// TIA Portal project "03_Montage_2018-09-26_KW" (V14)

(* hardware
DEVICE "S7300/ET200M-Station_4"  S7-300 station
   slot 0: "Profilschiene_0"  Rail  6ES7 390-1***0-0AA0
   slot 1: "PS 307 5A_1"  PS 307 5A  6ES7 307-1EA01-0AA0
   slot 2: "PLC_WBS_Bus"  CPU 314C-2 DP  6ES7 314-6CH04-0AB0  V3.3
      slot 0: "MPI-Schnittstelle_1"  MPI
      slot 1: "DP-Schnittstelle_1"  DP
      slot 2: "DI 24/DO 16_1"  DI24/DO16
      slot 3: "AI 5/AO 2_1"  AI5/AO2
      slot 4: "Zählen_1"  Counter
      slot 5: "Positionieren_1"  Positioning
   slot 4: "DI 64x24VDC sinking/souring_1"  DI64 x 24VDC  6ES7 321-1BP00-0AA0
   slot 5: "DI 64x24VDC sinking/souring_2"  DI64 x 24VDC  6ES7 321-1BP00-0AA0
   slot 6: "DI 64x24VDC sinking/souring_3"  DI64 x 24VDC  6ES7 321-1BP00-0AA0
   slot 7: "DI 64x24VDC sinking/souring_4"  DI64 x 24VDC  6ES7 321-1BP00-0AA0
   slot 8: "DO 64x24VDC/0.3A sourcing_1"  DO64 x 24VDC / 0.3A, P  6ES7 322-1BP00-0AA0
   slot 9: "DO 64x24VDC/0.3A sourcing_2"  DO64 x 24VDC / 0.3A, P  6ES7 322-1BP00-0AA0
   slot 10: "DO 64x24VDC/0.3A sourcing_3"  DO64 x 24VDC / 0.3A, P  6ES7 322-1BP00-0AA0
   slot 11: "DO 64x24VDC/0.3A sourcing_4"  DO64 x 24VDC / 0.3A, P  6ES7 322-1BP00-0AA0
*)

// ===== PLC "PLC_WBS_Bus"  CPU 314C-2 DP =====

VAR_GLOBAL   // PLC tag table "Standard-Variablentabelle"
   "Tag_1" AT %M20.0 : Bool;
   "Tag_2" AT %T0 : Timer;
END_VAR

VAR_GLOBAL   // PLC tag table "Betriebsart"
   "S0_HS" AT %E0.0 : Bool;   // Hauptschalter 0-Aus, 1-Ein
   "S1_Not_Halt" AT %E0.1 : Bool;   // Not-Halt NC
   "S2_START" AT %E0.2 : Bool;   // Taster START NO
   "S3_STOP" AT %E0.3 : Bool;   // Taster STOP NC
   "Res_E04" AT %E0.4 : Bool;
   "Res_E05" AT %E0.5 : Bool;
   "Res_E06" AT %E0.6 : Bool;
   "Res_E07" AT %E0.7 : Bool;
   "Res_E10" AT %E1.0 : Bool;
   "Res_E11" AT %E1.1 : Bool;
   "Res_E12" AT %E1.2 : Bool;
   "Res_E13" AT %E1.3 : Bool;
   "Res_E14" AT %E1.4 : Bool;
   "Res_E15" AT %E1.5 : Bool;
   "Res_E16" AT %E1.6 : Bool;
   "Factory_IO_RUN" AT %E1.7 : Bool;   // Rückmeldung Factory IO läuft
   "P1_MS_RT" AT %A0.0 : Bool;   // Meldesäule Rot
   "P2_MS_GE" AT %A0.1 : Bool;   // Meldesäule Gelb
   "P3_MS_GN" AT %A0.2 : Bool;   // Meldesäule Grün
   "P10_START" AT %A0.3 : Bool;   // Anzeige grün in START-Taster
   "P11_STOP" AT %A0.4 : Bool;   // Anzeige gelb in START-Taster
   "Res_A0.5" AT %A0.5 : Bool;
   "P12_Anfahrwarnung" AT %A0.6 : Bool;   // Rundumleuchte System
   "P13_Sirene" AT %A0.7 : Bool;   // Sirene System
   "Res_A10" AT %A1.0 : Bool;
   "Res_A11" AT %A1.1 : Bool;
   "Res_A12" AT %A1.2 : Bool;
   "Res_A13" AT %A1.3 : Bool;
   "Res_A14" AT %A1.4 : Bool;
   "Res_A15" AT %A1.5 : Bool;
   "Res_A16" AT %A1.6 : Bool;
   "Res_A17" AT %A1.7 : Bool;
   "Log_1" AT %M0.1 : Bool;   // statisch "1"
   "Log_0" AT %M0.0 : Bool;   // statisch "0"
   "Takt_1HZ" AT %M100.5 : Bool;   // Taktmerker 1 Hz
END_VAR

VAR_GLOBAL   // PLC tag table "Montage"
   "B3001_TB3001" AT %E2.0 : Bool;   // Transportband-Ende NC
   "B3002_TB3001" AT %E2.1 : Bool;   // Teil nachPositionierer NC
   "B3003_Teil_vor_POS" AT %E2.2 : Bool;   // Teil vor Positionierer NC
   "B3004_TB3001" AT %E2.3 : Bool;   // Transportband-Anfang NC
   "B3005_TB3002" AT %E2.4 : Bool;   // Transportband-Ende NC
   "B3006_TB3006" AT %E2.5 : Bool;   // Teil vor Schwenkarm NC
   "B3007_UT_BL" AT %E2.6 : Bool;   // Farbsensor Erkennung Farbteil Unterteil blau
   "B3008_OT_BL" AT %E2.7 : Bool;   // Farbsensor Erkennung Farbteil Oberteil blau
   "B3009_TB3006" AT %E3.0 : Bool;   // Transportband-Anfang NC
   "B3010_TB3007" AT %E3.1 : Bool;   // Transportband-Ende NC
   "B3011_TB3007" AT %E3.2 : Bool;   // Transportband-Anfang NC
   "B3012_TB3008" AT %E3.3 : Bool;   // Transportband-Ende NC
   "B3013_TB3008" AT %E3.4 : Bool;   // Transportband-Anfang NC
   "B3014_TB3005" AT %E3.5 : Bool;   // Transportband-Anfang NC
   "B3015_TB3005" AT %E3.6 : Bool;   // Transportband-Ende
   "B3016_TB3004" AT %E3.7 : Bool;   // Transportband-Anfang
   "B3017_Teil_vor_POS" AT %E4.0 : Bool;   // Teil vor Positionierer NC
   "B3018_TB3004" AT %E4.1 : Bool;   // Transportband-Ende NC
   "B3030_POS3001_geklemmt" AT %E4.2 : Bool;   // Positionierer RM geklemmt
   "B3031_POS3001_Heben_Senken" AT %E4.3 : Bool;   // Positionierer RM Bewegung
   "B3040_POS3002_geklemmt" AT %E4.4 : Bool;   // Positionierer RM geklemmt
   "B3041_POS3002_Heben_Senken" AT %E4.5 : Bool;   // Positionierer RM Bewegung
   "Res_E46" AT %E4.6 : Bool;
   "Res_E47" AT %E4.7 : Bool;
   "B3050_PAP3001_RM_X" AT %E5.0 : Bool;
   "B3051_PAP3001_RM_Z" AT %E5.1 : Bool;
   "B3052_PAP3001_Teil_erkannt" AT %E5.2 : Bool;
   "B3070_FZ_3001_Busy" AT %E5.3 : Bool;
   "B3071_FZ_3001_Error" AT %E5.4 : Bool;
   "B3072_FZ_Tür_offen" AT %E5.5 : Bool;
   "Res_E56" AT %E5.6 : Bool;
   "Res_E57" AT %E5.7 : Bool;
   "B4001_TB4001" AT %E6.0 : Bool;   // Transportband-Ende NC
   "B4002_TB4001" AT %E6.1 : Bool;   // Teil nachPositionierer NC
   "B4003_Teil_vor_POS" AT %E6.2 : Bool;   // Teil vor Positionierer NC
   "B4004_TB4001" AT %E6.3 : Bool;   // Transportband-Anfang NC
   "B4005_TB4002" AT %E6.4 : Bool;   // Transportband-Ende NC
   "B4006_TB4006" AT %E6.5 : Bool;   // Teil vor Schwenkarm NC
   "B4007_UT_GN" AT %E6.6 : Bool;   // Farbsensor Erkennung Farbteil Unterteil grün
   "B4008_OT_GN" AT %E6.7 : Bool;   // Farbsensor Erkennung Farbteil Oberteil grün
   "B4009_TB4006" AT %E7.0 : Bool;   // Transportband-Anfang NC
   "B4010_TB4007" AT %E7.1 : Bool;   // Transportband-Ende NC
   "B4011_TB4007" AT %E7.2 : Bool;   // Transportband-Anfang NC
   "B4012_TB4008" AT %E7.3 : Bool;   // Transportband-Ende NC
   "B4013_TB4008" AT %E7.4 : Bool;   // Transportband-Anfang NC
   "B4014_TB4005" AT %E7.5 : Bool;   // Transportband-Anfang NC
   "B4015_TB4005" AT %E7.6 : Bool;   // Transportband-Ende
   "B4016_TB4004" AT %E7.7 : Bool;   // Transportband-Anfang
   "B4017_Teil_vor_POS" AT %E8.0 : Bool;   // Teil vor Positionierer NC
   "B4018_TB4004" AT %E8.1 : Bool;   // Transportband-Ende NC
   "B4030_POS4001_geklemmt" AT %E8.2 : Bool;   // Positionierer RM geklemmt
   "B4031_POS4001_Heben_Senken" AT %E8.3 : Bool;   // Positionierer RM Bewegung
   "B4040_POS4002_geklemmt" AT %E8.4 : Bool;   // Positionierer RM geklemmt
   "B4041_POS4002_Heben_Senken" AT %E8.5 : Bool;   // Positionierer RM Bewegung
   "Res_E86" AT %E8.6 : Bool;
   "Res_E87" AT %E8.7 : Bool;
   "B4050_PAP4001_RM_X" AT %E9.0 : Bool;   // Pick-and-Place X-aktiv
   "B4051_PAP4001_RM_Z" AT %E9.1 : Bool;   // Pick-and-Place Z-aktiv
   "B4052_PAP4001_Teil_erkannt" AT %E9.2 : Bool;   // Teil am Greifer erkannt
   "B4070_FZ_4001_Busy" AT %E9.3 : Bool;   // Fertigungszentrum
   "B4071_FZ_4001_Error" AT %E9.4 : Bool;   // Fertigungszentrum
   "B4072_FZ_4001_Tür_offen" AT %E9.5 : Bool;   // Fertigungszentrum
   "Res_E96" AT %E9.6 : Bool;
   "Res_E97" AT %E9.7 : Bool;
   "TB3001" AT %A2.0 : Bool;
   "TB3002" AT %A2.1 : Bool;
   "TB3003" AT %A2.2 : Bool;
   "TB3004" AT %A2.3 : Bool;
   "TB3005" AT %A2.4 : Bool;
   "TB3006" AT %A2.5 : Bool;
   "TB3007" AT %A2.6 : Bool;
   "TB3008" AT %A2.7 : Bool;
   "FZ_3001_Start" AT %A3.0 : Bool;   // Fertigungszentrum Start
   "FZ_3001_Stop" AT %A3.1 : Bool;   // Fertigungszentrum Stop
   "FZ_3001_OT_UT" AT %A3.2 : Bool;   // Fertigungszentrum UT =0 / OT=1
   "Sorter_Arm_3001_schwenken" AT %A3.3 : Bool;
   "Sorter_Arm_3001_Band_V" AT %A3.4 : Bool;
   "Sorter_Arm_3001_Band_R" AT %A3.5 : Bool;
   "POS3001_Klemmen" AT %A3.6 : Bool;
   "POS3001_Heben" AT %A3.7 : Bool;
   "POS3002_Klemmen" AT %A4.0 : Bool;
   "POS3002_Heben" AT %A4.1 : Bool;
   "PAP3001_X" AT %A4.2 : Bool;
   "PAP3001_Z" AT %A4.3 : Bool;
   "PAP3001_Greifer" AT %A4.4 : Bool;
   "STOP_3001" AT %A4.5 : Bool;
   "Res_A46" AT %A4.6 : Bool;
   "Emitter_1" AT %A4.7 : Bool;
   "TB4001" AT %A5.0 : Bool;
   "TB4002" AT %A5.1 : Bool;
   "TB4003" AT %A5.2 : Bool;
   "TB4004" AT %A5.3 : Bool;
   "TB4005" AT %A5.4 : Bool;
   "TB4006" AT %A5.5 : Bool;
   "TB4007" AT %A5.6 : Bool;
   "TB4008" AT %A5.7 : Bool;
   "FZ_4001_Start" AT %A6.0 : Bool;   // Fertigungszentrum Start
   "FZ_4001_Stop" AT %A6.1 : Bool;   // Fertigungszentrum Stop
   "FZ_4001_OT_UT" AT %A6.2 : Bool;   // Fertigungszentrum UT =0 / OT=1
   "Sorter_Arm_4001_schwenken" AT %A6.3 : Bool;
   "Sorter_Arm_4001_Band_V" AT %A6.4 : Bool;
   "Sorter_Arm_4001_Band_R" AT %A6.5 : Bool;
   "POS4001_Klemmen" AT %A6.6 : Bool;
   "POS4001_Heben" AT %A6.7 : Bool;
   "POS4002_Klemmen" AT %A7.0 : Bool;
   "POS4002_Heben" AT %A7.1 : Bool;
   "PAP4001_X" AT %A7.2 : Bool;
   "PAP4001_Z" AT %A7.3 : Bool;
   "PAP4001_Greifer" AT %A7.4 : Bool;
   "STOP4001" AT %A7.5 : Bool;
   "Res_A76" AT %A7.6 : Bool;
   "Emitter_2" AT %A7.7 : Bool;
   "FZ_3001_Bearbeitungszeit" AT %EW20 : Int;
   "FZ_4001_Bearbeitungszeit" AT %EW22 : Int;
END_VAR

VAR_GLOBAL   // PLC tag table "KW"
   "Anlage_Start" AT %M22.0 : Bool;
   "Freigabe_Start" AT %M22.1 : Bool;
   "M_HOT_HALT" AT %M22.2 : Bool;
   "FLK_S2_Start" AT %M22.3 : Bool;
   "B1_Freigabe" AT %M22.4 : Bool;
   "Teile_Typ" AT %M22.5 : Bool;
   "FLK_B4010_TB4007" AT %M22.6 : Bool;
   "FreiFürTB4006" AT %M22.7 : Bool;
   "UT_an_Weiche" AT %M23.0 : Bool;
   "OT_an_Weiche" AT %M23.1 : Bool;
   "FreiFürTB4005" AT %M23.2 : Bool;
   "Glob_Sperre" AT %M23.3 : Bool;
   "FreiFürTB4002" AT %M23.4 : Bool;
   "M_Entklemmen" AT %M23.5 : Bool;
   "03_M_OT_Abfuehren" AT %M23.6 : Bool;
   "03_M_UT_Abfuehren" AT %M23.7 : Bool;
   "MT_OT_Bereit" AT %M24.0 : Bool;
   "MT_UT_Bereit" AT %M24.1 : Bool;
   "03_GRN_OT_det" AT %M24.2 : Bool;
   "03_GRN_UT_det" AT %M24.3 : Bool;
   "03_BLAU_OT_det" AT %M24.4 : Bool;
   "03_BLAU_UT_det" AT %M24.5 : Bool;
   "03_GRN_FRGB_CNC" AT %M24.6 : Bool;
   "03_BLAU_FRGB_CNC" AT %M24.7 : Bool;
   "03_GRN_CNC_MTR_AN" AT %M25.0 : Bool;
   "03_BLAU_CNC_MTR_AN" AT %M25.1 : Bool;
   "delete_1" AT %M25.2 : Bool;
   "delete_2" AT %M25.3 : Bool;
   "03_GRN_OT_FRG" AT %M25.4 : Bool;
   "03_GRN_UT_FRG" AT %M25.5 : Bool;
   "03_BLAU_OT_FRG" AT %M25.6 : Bool;
   "03_BLAU_UT_FRG" AT %M25.7 : Bool;
END_VAR

DATA_BLOCK "03_04-OT_Grueneteile"   // DB2
{ S7_Optimized_Access := 'FALSE' }
VERSION : 0.1
// stored: InstanceOfName Foerderband_m_Klemme
"Foerderband_m_Klemme"
BEGIN
END_DATA_BLOCK

DATA_BLOCK "03_04_UT_Grueneteile"   // DB3
{ S7_Optimized_Access := 'FALSE' }
VERSION : 0.1
// stored: InstanceOfName Foerderband_m_Klemme
"Foerderband_m_Klemme"
BEGIN
END_DATA_BLOCK

DATA_BLOCK "03_04_PnP_Grueneteile"   // DB4
{ S7_Optimized_Access := 'FALSE' }
VERSION : 0.1
// stored: InstanceOfName Pick_n_Place
"Pick_n_Place"
BEGIN
END_DATA_BLOCK

DATA_BLOCK "03_04_MNTG_Grueneteile"   // DB5
{ S7_Optimized_Access := 'FALSE' }
VERSION : 0.1
// stored: InstanceOfName 03_04_MNTG_BL
"03_04_MNTG_BL"
BEGIN
END_DATA_BLOCK

DATA_BLOCK "03_04_MNTG_Blaueteile"   // DB6
{ S7_Optimized_Access := 'FALSE' }
VERSION : 0.1
// stored: InstanceOfName 03_04_MNTG_BL
"03_04_MNTG_BL"
BEGIN
END_DATA_BLOCK

DATA_BLOCK "03_04-OT_Blaueteile"   // DB7
{ S7_Optimized_Access := 'FALSE' }
VERSION : 0.1
// stored: InstanceOfName Foerderband_m_Klemme
"Foerderband_m_Klemme"
BEGIN
END_DATA_BLOCK

DATA_BLOCK "03_04_UT_Blaueteile"   // DB8
{ S7_Optimized_Access := 'FALSE' }
VERSION : 0.1
// stored: InstanceOfName Foerderband_m_Klemme
"Foerderband_m_Klemme"
BEGIN
END_DATA_BLOCK

DATA_BLOCK "03_04_PnP_Blaueteile"   // DB9
{ S7_Optimized_Access := 'FALSE' }
VERSION : 0.1
// stored: InstanceOfName Pick_n_Place
"Pick_n_Place"
BEGIN
END_DATA_BLOCK

DATA_BLOCK "FB_OT_Gruen"   // DB10
{ S7_Optimized_Access := 'FALSE' }
VERSION : 0.1
// stored: InstanceOfName Foerderband_m_Klemme
"Foerderband_m_Klemme"
BEGIN
END_DATA_BLOCK

DATA_BLOCK "FB_UT_Gruen"   // DB11
{ S7_Optimized_Access := 'FALSE' }
VERSION : 0.1
// stored: InstanceOfName Foerderband_m_Klemme
"Foerderband_m_Klemme"
BEGIN
END_DATA_BLOCK

DATA_BLOCK "03_01_Grueneteile"   // DB12
{ S7_Optimized_Access := 'FALSE' }
VERSION : 0.1
// stored: InstanceOfName 03_01_Anlaufbaender
"03_01_Anlaufbaender"
BEGIN
END_DATA_BLOCK

DATA_BLOCK "03_01_Blaueteile"   // DB13
{ S7_Optimized_Access := 'FALSE' }
VERSION : 0.1
// stored: InstanceOfName 03_01_Anlaufbaender
"03_01_Anlaufbaender"
BEGIN
END_DATA_BLOCK

DATA_BLOCK "03_02_Grueneteile"   // DB14
{ S7_Optimized_Access := 'FALSE' }
VERSION : 0.1
// stored: InstanceOfName 03_02_Bearbeitungszelle
"03_02_Bearbeitungszelle"
BEGIN
END_DATA_BLOCK

DATA_BLOCK "03_02_Blaueteile"   // DB15
{ S7_Optimized_Access := 'FALSE' }
VERSION : 0.1
// stored: InstanceOfName 03_02_Bearbeitungszelle
"03_02_Bearbeitungszelle"
BEGIN
END_DATA_BLOCK

DATA_BLOCK "03_03_Grueneteile"   // DB16
{ S7_Optimized_Access := 'FALSE' }
VERSION : 0.1
// stored: InstanceOfName 03_03_Weiche
"03_03_Weiche"
BEGIN
END_DATA_BLOCK

DATA_BLOCK "03_03_Blaueteile"   // DB17
{ S7_Optimized_Access := 'FALSE' }
VERSION : 0.1
// stored: InstanceOfName 03_03_Weiche
"03_03_Weiche"
BEGIN
END_DATA_BLOCK

DATA_BLOCK "PnP_Gruen"   // DB18
{ S7_Optimized_Access := 'FALSE' }
VERSION : 0.1
// stored: InstanceOfName Pick_n_Place
"Pick_n_Place"
BEGIN
END_DATA_BLOCK

DATA_BLOCK "03_04_MNTG_GR_DB"   // DB19
{ S7_Optimized_Access := 'FALSE' }
VERSION : 0.1
// stored: InstanceOfName 03_04_MNTG_GR
"03_04_MNTG_GR"
BEGIN
END_DATA_BLOCK

FUNCTION_BLOCK "03_04_MNTG_BL"   // FB1, FBD
{ S7_Optimized_Access := 'FALSE' }
VERSION : 0.1
   VAR_OUTPUT
      OT_Freigabe : Bool;
      UT_Freigabe : Bool;
   END_VAR
   VAR
      OT_angesaugt : Bool;
      OT_losgelassen : Bool;
      OT_Band : "Foerderband_m_Klemme";
      UT_Band : "Foerderband_m_Klemme";
      PicknPlace : "Pick_n_Place";
   END_VAR
BEGIN

REGION Network 1: BLAU OT Klemm-Foerderband
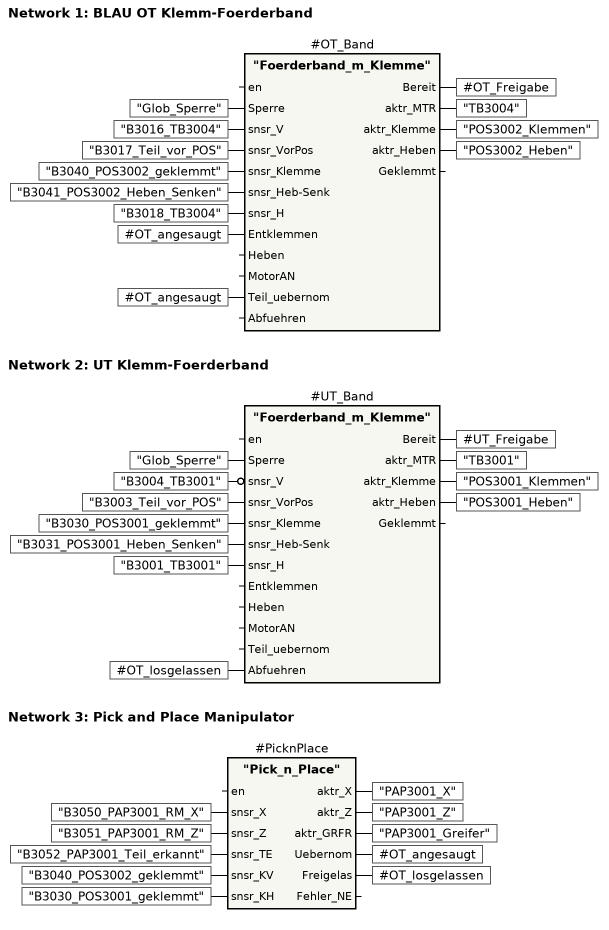
   #OT_Band(Sperre := "Glob_Sperre",   // "Foerderband_m_Klemme"
            snsr_V := "B3016_TB3004",
            snsr_VorPos := "B3017_Teil_vor_POS",
            snsr_Klemme := "B3040_POS3002_geklemmt",
            "snsr_Heb-Senk" := "B3041_POS3002_Heben_Senken",
            snsr_H := "B3018_TB3004",
            Entklemmen := #OT_angesaugt,
            Teil_uebernom := #OT_angesaugt,
            Bereit => #OT_Freigabe,
            aktr_MTR => "TB3004",
            aktr_Klemme => "POS3002_Klemmen",
            aktr_Heben => "POS3002_Heben");
END_REGION

REGION Network 2: UT Klemm-Foerderband
   #UT_Band(Sperre := "Glob_Sperre",   // "Foerderband_m_Klemme"
            snsr_V := NOT "B3004_TB3001",
            snsr_VorPos := "B3003_Teil_vor_POS",
            snsr_Klemme := "B3030_POS3001_geklemmt",
            "snsr_Heb-Senk" := "B3031_POS3001_Heben_Senken",
            snsr_H := "B3001_TB3001",
            Abfuehren := #OT_losgelassen,
            Bereit => #UT_Freigabe,
            aktr_MTR => "TB3001",
            aktr_Klemme => "POS3001_Klemmen",
            aktr_Heben => "POS3001_Heben");
END_REGION

REGION Network 3: Pick and Place Manipulator
   #PicknPlace(snsr_X := "B3050_PAP3001_RM_X",   // "Pick_n_Place"
               snsr_Z := "B3051_PAP3001_RM_Z",
               snsr_TE := "B3052_PAP3001_Teil_erkannt",
               snsr_KV := "B3040_POS3002_geklemmt",
               snsr_KH := "B3030_POS3001_geklemmt",
               aktr_X => "PAP3001_X",
               aktr_Z => "PAP3001_Z",
               aktr_GRFR => "PAP3001_Greifer",
               Uebernom => #OT_angesaugt,
               Freigelas => #OT_losgelassen);
END_REGION
END_FUNCTION_BLOCK

FUNCTION_BLOCK "03_04_MNTG_GR"   // FB2, FBD
{ S7_Optimized_Access := 'FALSE' }
VERSION : 0.1
   VAR_OUTPUT
      OT_Freigabe : Bool;
      UT_Freigabe : Bool;
   END_VAR
   VAR
      OT_Band_DB : "Foerderband_m_Klemme";
      UT_Band_DB : "Foerderband_m_Klemme";
      PnP_DB : "Pick_n_Place";
      OT_angesaugt : Bool;
      OT_losgelassen : Bool;
   END_VAR
BEGIN

REGION Network 1: GRUEN OT Klemm-Foerderband
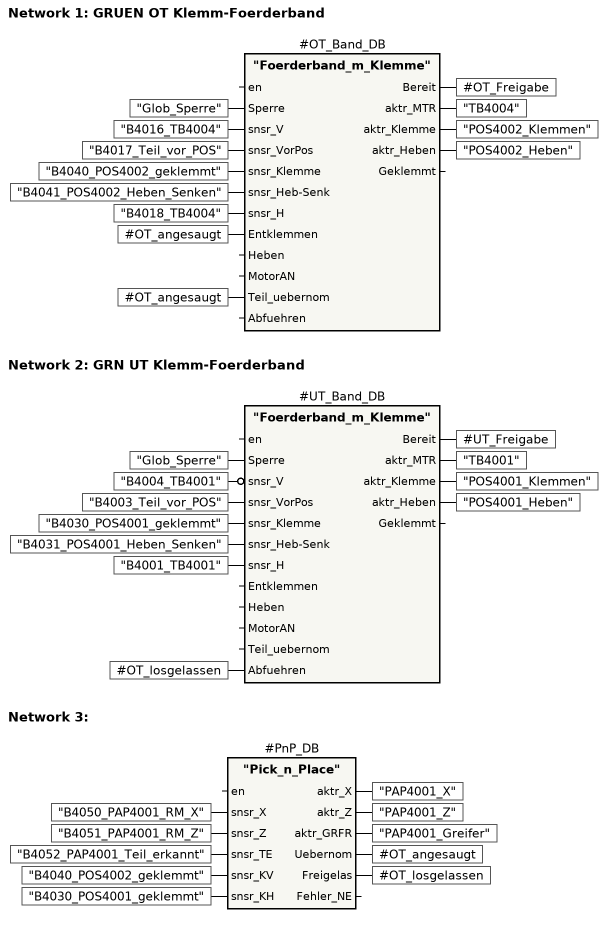
   #OT_Band_DB(Sperre := "Glob_Sperre",   // "Foerderband_m_Klemme"
               snsr_V := "B4016_TB4004",
               snsr_VorPos := "B4017_Teil_vor_POS",
               snsr_Klemme := "B4040_POS4002_geklemmt",
               "snsr_Heb-Senk" := "B4041_POS4002_Heben_Senken",
               snsr_H := "B4018_TB4004",
               Entklemmen := #OT_angesaugt,
               Teil_uebernom := #OT_angesaugt,
               Bereit => #OT_Freigabe,
               aktr_MTR => "TB4004",
               aktr_Klemme => "POS4002_Klemmen",
               aktr_Heben => "POS4002_Heben");
END_REGION

REGION Network 2: GRN UT Klemm-Foerderband
   #UT_Band_DB(Sperre := "Glob_Sperre",   // "Foerderband_m_Klemme"
               snsr_V := NOT "B4004_TB4001",
               snsr_VorPos := "B4003_Teil_vor_POS",
               snsr_Klemme := "B4030_POS4001_geklemmt",
               "snsr_Heb-Senk" := "B4031_POS4001_Heben_Senken",
               snsr_H := "B4001_TB4001",
               Abfuehren := #OT_losgelassen,
               Bereit => #UT_Freigabe,
               aktr_MTR => "TB4001",
               aktr_Klemme => "POS4001_Klemmen",
               aktr_Heben => "POS4001_Heben");
END_REGION

REGION Network 3
   #PnP_DB(snsr_X := "B4050_PAP4001_RM_X",   // "Pick_n_Place"
           snsr_Z := "B4051_PAP4001_RM_Z",
           snsr_TE := "B4052_PAP4001_Teil_erkannt",
           snsr_KV := "B4040_POS4002_geklemmt",
           snsr_KH := "B4030_POS4001_geklemmt",
           aktr_X => "PAP4001_X",
           aktr_Z => "PAP4001_Z",
           aktr_GRFR => "PAP4001_Greifer",
           Uebernom => #OT_angesaugt,
           Freigelas => #OT_losgelassen);
END_REGION
END_FUNCTION_BLOCK

FUNCTION_BLOCK "Foerderband_m_Klemme"   // FB3, LAD
{ S7_Optimized_Access := 'FALSE' }
VERSION : 0.1
   VAR_INPUT
      Sperre : Bool;
      snsr_V : Bool;   // (NC) =1 wenn betätigt
      snsr_VorPos : Bool;   // (NO) =0 wenn betätigt
      snsr_Klemme : Bool;   // (NC) =1 wenn betätigt
      "snsr_Heb-Senk" : Bool;   // (NO) =0 wenn betätigt
      snsr_H : Bool;   // (NO) =0 wenn betätigt
      Entklemmen : Bool;   // =1 entklemmen
      Heben : Bool;   // =0 unten, =1 oben
      MotorAN : Bool;   // =1 Motor AN, =0 Motor AUS
      Teil_uebernom : Bool;   // =0 passiv, =1 aktiv
   END_VAR
   VAR_OUTPUT
      Bereit : Bool;
      aktr_MTR : Bool;
      aktr_Klemme : Bool;
      aktr_Heben : Bool;
      Geklemmt : Bool;
   END_VAR
   VAR_IN_OUT
      Abfuehren : Bool;
   END_VAR
   VAR
      Beladen : Bool;
      FLK_Letzter_Sensor : Bool;
      "FLK_Vor-Pos" : Bool;
      LetSens_P_Flanke : Bool;
      Abfuhr_Modus : Bool;
   END_VAR
   VAR_TEMP   // added for the SCL form of the ladder/FBD networks
      _w1 : Bool;
   END_VAR
BEGIN

REGION Network 1: Letzter Sensor positive Flankenerkennung
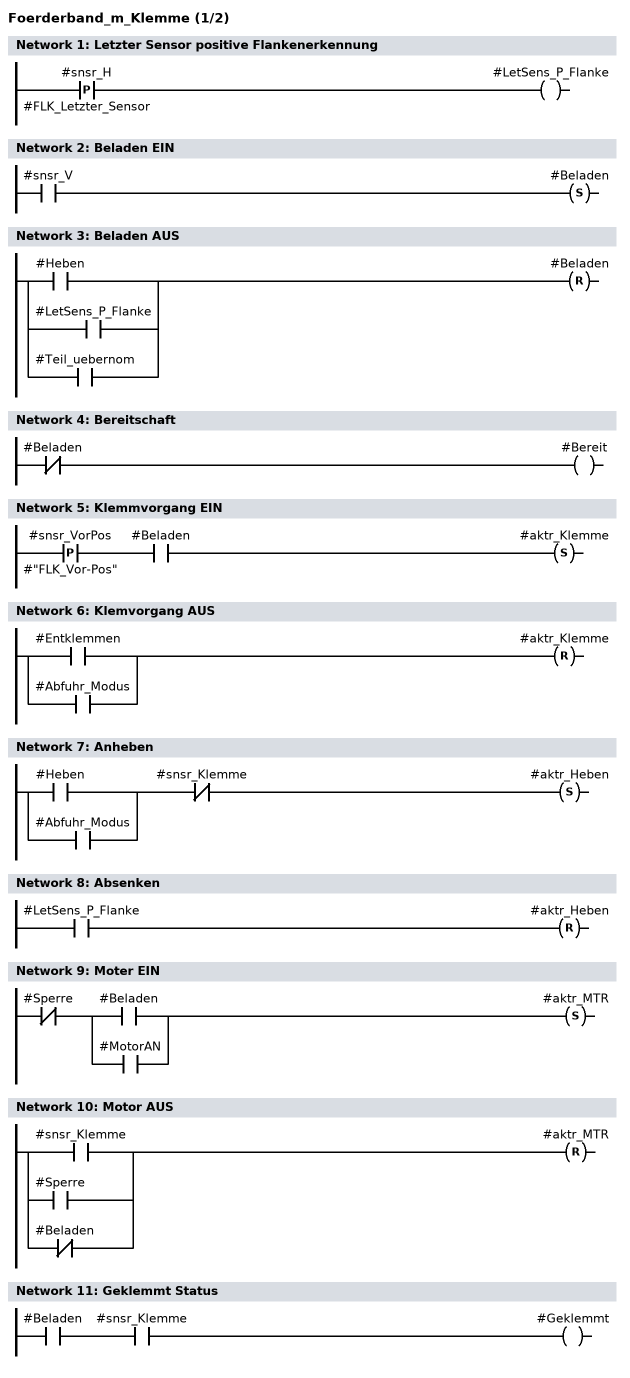
   RUNG wire#powerrail
      P_Contact(operand := #snsr_H, bit := #FLK_Letzter_Sensor)
      Coil( #LetSens_P_Flanke )
   END_RUNG
   // the same network as SCL:
   #_w1 := #snsr_H AND NOT #FLK_Letzter_Sensor;   // rising edge of #snsr_H
   #FLK_Letzter_Sensor := #snsr_H;
   #LetSens_P_Flanke := #_w1;
END_REGION

REGION Network 2: Beladen EIN
   RUNG wire#powerrail
      Contact( #snsr_V )
      S_Coil( #Beladen )
   END_RUNG
   // the same network as SCL:
   IF #snsr_V THEN #Beladen := TRUE; END_IF;
END_REGION

REGION Network 3: Beladen AUS
   RUNG wire#powerrail
      Contact( #Heben )
      wire#w1
      R_Coil( #Beladen )
   END_RUNG
   RUNG wire#powerrail
      Contact( #LetSens_P_Flanke )
   END_RUNG wire#w1
   RUNG wire#powerrail
      Contact( #Teil_uebernom )
   END_RUNG wire#w1
   // the same network as SCL:
   IF #Heben OR #LetSens_P_Flanke OR #Teil_uebernom THEN #Beladen := FALSE; END_IF;
END_REGION

REGION Network 4: Bereitschaft
   RUNG wire#powerrail
      I_Contact( #Beladen )
      Coil( #Bereit )
   END_RUNG
   // the same network as SCL:
   #Bereit := NOT #Beladen;
END_REGION

REGION Network 5: Klemmvorgang EIN
   RUNG wire#powerrail
      P_Contact(operand := #snsr_VorPos, bit := #"FLK_Vor-Pos")
      Contact( #Beladen )
      S_Coil( #aktr_Klemme )
   END_RUNG
   // the same network as SCL:
   #_w1 := #snsr_VorPos AND NOT #"FLK_Vor-Pos";   // rising edge of #snsr_VorPos
   #"FLK_Vor-Pos" := #snsr_VorPos;
   IF #_w1 AND #Beladen THEN #aktr_Klemme := TRUE; END_IF;
END_REGION

REGION Network 6: Klemvorgang AUS
   RUNG wire#powerrail
      Contact( #Entklemmen )
      wire#w1
      R_Coil( #aktr_Klemme )
   END_RUNG
   RUNG wire#powerrail
      Contact( #Abfuhr_Modus )
   END_RUNG wire#w1
   // the same network as SCL:
   IF #Entklemmen OR #Abfuhr_Modus THEN #aktr_Klemme := FALSE; END_IF;
END_REGION

REGION Network 7: Anheben
   RUNG wire#powerrail
      Contact( #Heben )
      wire#w1
      I_Contact( #snsr_Klemme )
      S_Coil( #aktr_Heben )
   END_RUNG
   RUNG wire#powerrail
      Contact( #Abfuhr_Modus )
   END_RUNG wire#w1
   // the same network as SCL:
   IF (#Heben OR #Abfuhr_Modus) AND NOT #snsr_Klemme THEN #aktr_Heben := TRUE; END_IF;
END_REGION

REGION Network 8: Absenken
   RUNG wire#powerrail
      Contact( #LetSens_P_Flanke )
      R_Coil( #aktr_Heben )
   END_RUNG
   // the same network as SCL:
   IF #LetSens_P_Flanke THEN #aktr_Heben := FALSE; END_IF;
END_REGION

REGION Network 9: Moter EIN
   RUNG wire#powerrail
      I_Contact( #Sperre )
      wire#w1
      Contact( #Beladen )
      wire#w2
      S_Coil( #aktr_MTR )
   END_RUNG
   RUNG wire#w1
      Contact( #MotorAN )
   END_RUNG wire#w2
   // the same network as SCL:
   IF NOT #Sperre AND (#Beladen OR #MotorAN) THEN #aktr_MTR := TRUE; END_IF;
END_REGION

REGION Network 10: Motor AUS
   RUNG wire#powerrail
      Contact( #snsr_Klemme )
      wire#w1
      R_Coil( #aktr_MTR )
   END_RUNG
   RUNG wire#powerrail
      Contact( #Sperre )
   END_RUNG wire#w1
   RUNG wire#powerrail
      I_Contact( #Beladen )
   END_RUNG wire#w1
   // the same network as SCL:
   IF #snsr_Klemme OR #Sperre OR NOT #Beladen THEN #aktr_MTR := FALSE; END_IF;
END_REGION

REGION Network 11: Geklemmt Status
   RUNG wire#powerrail
      Contact( #Beladen )
      Contact( #snsr_Klemme )
      Coil( #Geklemmt )
   END_RUNG
   // the same network as SCL:
   #Geklemmt := #Beladen AND #snsr_Klemme;
END_REGION

REGION Network 12: SR Abfuhr_Modus
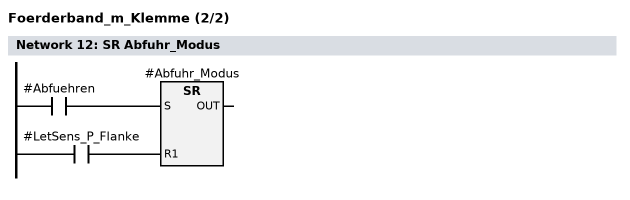
   RUNG wire#powerrail
      Contact( #Abfuehren )
      S_SR(operand := #Abfuhr_Modus, r1 := wire#w1)
   END_RUNG
   RUNG wire#powerrail
      Contact( #LetSens_P_Flanke )
   END_RUNG wire#w1
   // the same network as SCL:
   IF #Abfuehren THEN
       #Abfuhr_Modus := TRUE;   // SR flip-flop
   END_IF;
   IF #LetSens_P_Flanke THEN #Abfuhr_Modus := FALSE; END_IF;
END_REGION
END_FUNCTION_BLOCK

FUNCTION_BLOCK "03_01_Anlaufbaender"   // FB4, LAD
{ S7_Optimized_Access := 'FALSE' }
VERSION : 0.1
   VAR_INPUT
      snsr_V1 : Bool;
      snsr_V2 : Bool;
      snsr_H1 : Bool;
      snsr_H2 : Bool;
      Freigabe_IN : Bool;
      Sperre : Bool;
   END_VAR
   VAR_OUTPUT
      aktr_MTR_1 : Bool;
      aktr_MTR_2 : Bool;
      Freigabe_OUT : Bool;
   END_VAR
   VAR
      Beladen_1 : Bool;
      Beladen_2 : Bool;
      FLK_H1 : Bool;
      FLK_H2 : Bool;
   END_VAR
   VAR_TEMP   // added for the SCL form of the ladder/FBD networks
      _w1 : Bool;
   END_VAR
BEGIN

REGION Network 1: Reset Beladen_1
   // Reset des Statuses BELADEN der ersten Förderband
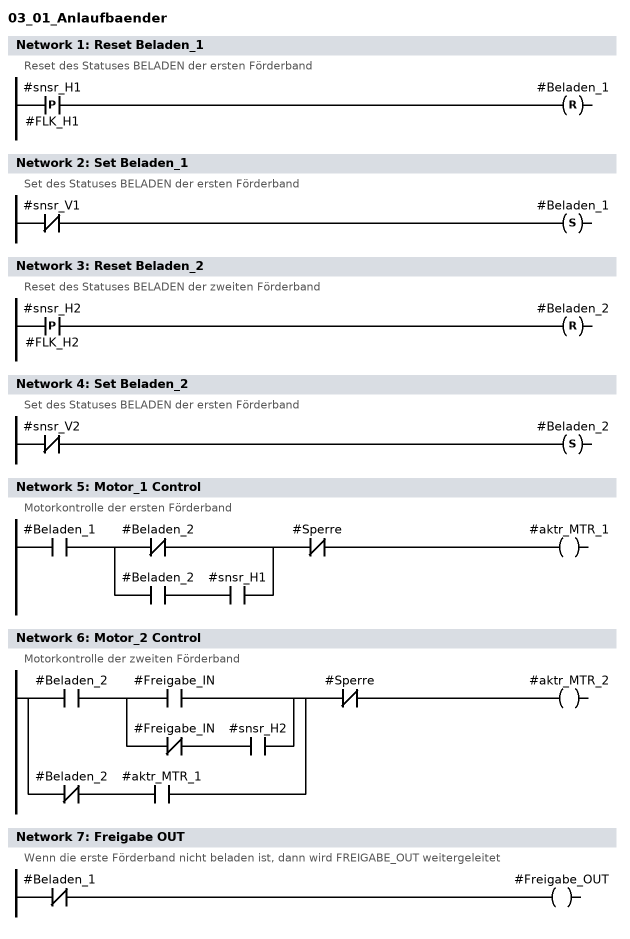
   RUNG wire#powerrail
      P_Contact(operand := #snsr_H1, bit := #FLK_H1)
      R_Coil( #Beladen_1 )
   END_RUNG
   // the same network as SCL:
   #_w1 := #snsr_H1 AND NOT #FLK_H1;   // rising edge of #snsr_H1
   #FLK_H1 := #snsr_H1;
   IF #_w1 THEN #Beladen_1 := FALSE; END_IF;
END_REGION

REGION Network 2: Set Beladen_1
   // Set des Statuses BELADEN der ersten Förderband
   RUNG wire#powerrail
      I_Contact( #snsr_V1 )
      S_Coil( #Beladen_1 )
   END_RUNG
   // the same network as SCL:
   IF NOT #snsr_V1 THEN #Beladen_1 := TRUE; END_IF;
END_REGION

REGION Network 3: Reset Beladen_2
   // Reset des Statuses BELADEN der zweiten Förderband
   RUNG wire#powerrail
      P_Contact(operand := #snsr_H2, bit := #FLK_H2)
      R_Coil( #Beladen_2 )
   END_RUNG
   // the same network as SCL:
   #_w1 := #snsr_H2 AND NOT #FLK_H2;   // rising edge of #snsr_H2
   #FLK_H2 := #snsr_H2;
   IF #_w1 THEN #Beladen_2 := FALSE; END_IF;
END_REGION

REGION Network 4: Set Beladen_2
   // Set des Statuses BELADEN der ersten Förderband
   RUNG wire#powerrail
      I_Contact( #snsr_V2 )
      S_Coil( #Beladen_2 )
   END_RUNG
   // the same network as SCL:
   IF NOT #snsr_V2 THEN #Beladen_2 := TRUE; END_IF;
END_REGION

REGION Network 5: Motor_1 Control
   // Motorkontrolle der ersten Förderband
   RUNG wire#powerrail
      Contact( #Beladen_1 )
      wire#w1
      I_Contact( #Beladen_2 )
      wire#w2
      I_Contact( #Sperre )
      Coil( #aktr_MTR_1 )
   END_RUNG
   RUNG wire#w1
      Contact( #Beladen_2 )
      Contact( #snsr_H1 )
   END_RUNG wire#w2
   // the same network as SCL:
   #aktr_MTR_1 := #Beladen_1 AND (NOT #Beladen_2 OR (#Beladen_2 AND #snsr_H1)) AND NOT #Sperre;
END_REGION

REGION Network 6: Motor_2 Control
   // Motorkontrolle der zweiten Förderband
   RUNG wire#powerrail
      Contact( #Beladen_2 )
      wire#w1
      Contact( #Freigabe_IN )
      wire#w2
      I_Contact( #Sperre )
      Coil( #aktr_MTR_2 )
   END_RUNG
   RUNG wire#w1
      I_Contact( #Freigabe_IN )
      Contact( #snsr_H2 )
   END_RUNG wire#w2
   RUNG wire#powerrail
      I_Contact( #Beladen_2 )
      Contact( #aktr_MTR_1 )
   END_RUNG wire#w2
   // the same network as SCL:
   #aktr_MTR_2 := ((#Beladen_2 AND (#Freigabe_IN OR (NOT #Freigabe_IN AND #snsr_H2))) OR (NOT #Beladen_2 AND #aktr_MTR_1)) AND NOT #Sperre;
END_REGION

REGION Network 7: Freigabe OUT
   // Wenn die erste Förderband nicht beladen ist, dann wird FREIGABE_OUT weitergeleitet
   RUNG wire#powerrail
      I_Contact( #Beladen_1 )
      Coil( #Freigabe_OUT )
   END_RUNG
   // the same network as SCL:
   #Freigabe_OUT := NOT #Beladen_1;
END_REGION
END_FUNCTION_BLOCK

FUNCTION_BLOCK "Pick_n_Place"   // FB5, LAD
TITLE = Montage Pick_n_Place
{ S7_Optimized_Access := 'FALSE' }
VERSION : 0.1
   VAR_INPUT
      snsr_X : Bool;
      snsr_Z : Bool;
      snsr_TE : Bool;
      snsr_KV : Bool;
      snsr_KH : Bool;
   END_VAR
   VAR_OUTPUT
      aktr_X : Bool;
      aktr_Z : Bool;
      aktr_GRFR : Bool;
      Uebernom : Bool;
      Freigelas : Bool;
      Fehler_NE : Bool;
   END_VAR
   VAR
      X0 : Bool;
      X1 : Bool;
      X2 : Bool;
      X3 : Bool;
      X4 : Bool;
      X5 : Bool;
      X6 : Bool;
      X7 : Bool;
      X8 : Bool;
      X9 : Bool;
      IF_X1 : Bool;
      IF_X2 : Bool;
      IF_X3 : Bool;
      IF_X4 : Bool;
      IF_X5 : Bool;
      IF_X6 : Bool;
      IF_X7 : Bool;
      IF_X8 : Bool;
      IF_X9 : Bool;
      flk_X1 : Bool;
      flk_X2 : Bool;
      flk_X3 : Bool;
      flk_X4 : Bool;
      flk_X5 : Bool;
      flk_X6 : Bool;
      flk_X7 : Bool;
      flk_X8 : Bool;
      flk_X9 : Bool;
      Zmove_ended : Bool;
      Xmove_ended : Bool;
      flk_Xmove : Bool;
      flk_Zmove : Bool;
   END_VAR
   VAR_TEMP   // added for the SCL form of the ladder/FBD networks
      _w1 : Bool;
   END_VAR
BEGIN

REGION Network 1: Grundstellung
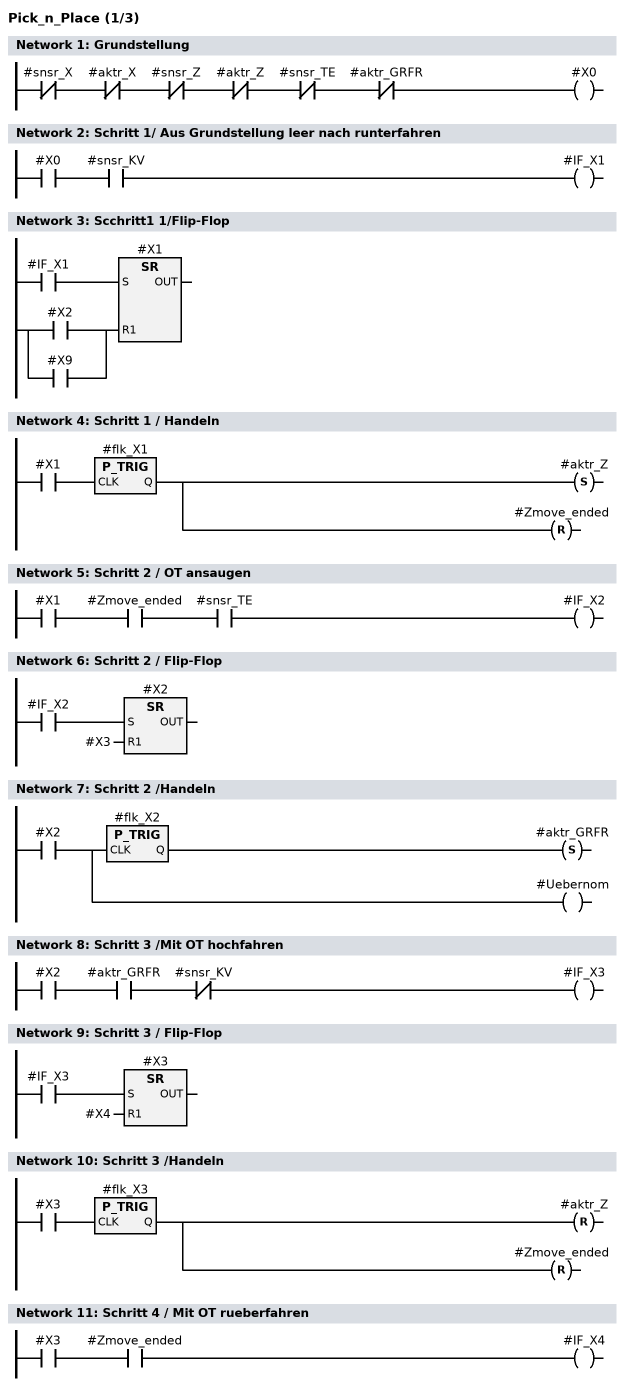
   RUNG wire#powerrail
      I_Contact( #snsr_X )
      I_Contact( #aktr_X )
      I_Contact( #snsr_Z )
      I_Contact( #aktr_Z )
      I_Contact( #snsr_TE )
      I_Contact( #aktr_GRFR )
      Coil( #X0 )
   END_RUNG
   // the same network as SCL:
   #X0 := NOT #snsr_X AND NOT #aktr_X AND NOT #snsr_Z AND NOT #aktr_Z AND NOT #snsr_TE AND NOT #aktr_GRFR;
END_REGION

REGION Network 2: Schritt 1/ Aus Grundstellung leer nach runterfahren
   RUNG wire#powerrail
      Contact( #X0 )
      Contact( #snsr_KV )
      Coil( #IF_X1 )
   END_RUNG
   // the same network as SCL:
   #IF_X1 := #X0 AND #snsr_KV;
END_REGION

REGION Network 3: Scchritt1 1/Flip-Flop
   RUNG wire#powerrail
      Contact( #IF_X1 )
      S_SR(operand := #X1, r1 := wire#w1)
   END_RUNG
   RUNG wire#powerrail
      Contact( #X2 )
   END_RUNG wire#w1
   RUNG wire#powerrail
      Contact( #X9 )
   END_RUNG wire#w1
   // the same network as SCL:
   IF #IF_X1 THEN
       #X1 := TRUE;   // SR flip-flop
   END_IF;
   IF #X2 OR #X9 THEN #X1 := FALSE; END_IF;
END_REGION

REGION Network 4: Schritt 1 / Handeln
   RUNG wire#powerrail
      Contact( #X1 )
      P_Trig( #flk_X1 )
      wire#w1
      S_Coil( #aktr_Z )
   END_RUNG
   RUNG wire#w1
      R_Coil( #Zmove_ended )
   END_RUNG
   // the same network as SCL:
   #_w1 := #X1 AND NOT #flk_X1;   // rising edge
   #flk_X1 := #X1;
   IF #_w1 THEN
       #aktr_Z := TRUE;
       #Zmove_ended := FALSE;
   END_IF;
END_REGION

REGION Network 5: Schritt 2 / OT ansaugen
   RUNG wire#powerrail
      Contact( #X1 )
      Contact( #Zmove_ended )
      Contact( #snsr_TE )
      Coil( #IF_X2 )
   END_RUNG
   // the same network as SCL:
   #IF_X2 := #X1 AND #Zmove_ended AND #snsr_TE;
END_REGION

REGION Network 6: Schritt 2 / Flip-Flop
   RUNG wire#powerrail
      Contact( #IF_X2 )
      S_SR(operand := #X2, r1 := #X3)
   END_RUNG
   // the same network as SCL:
   IF #IF_X2 THEN
       #X2 := TRUE;   // SR flip-flop
   END_IF;
   IF #X3 THEN #X2 := FALSE; END_IF;
END_REGION

REGION Network 7: Schritt 2 /Handeln
   RUNG wire#powerrail
      Contact( #X2 )
      wire#w1
      P_Trig( #flk_X2 )
      S_Coil( #aktr_GRFR )
   END_RUNG
   RUNG wire#w1
      Coil( #Uebernom )
   END_RUNG
   // the same network as SCL:
   #_w1 := #X2 AND NOT #flk_X2;   // rising edge
   #flk_X2 := #X2;
   IF #_w1 THEN #aktr_GRFR := TRUE; END_IF;
   #Uebernom := #X2;
END_REGION

REGION Network 8: Schritt 3 /Mit OT hochfahren
   RUNG wire#powerrail
      Contact( #X2 )
      Contact( #aktr_GRFR )
      I_Contact( #snsr_KV )
      Coil( #IF_X3 )
   END_RUNG
   // the same network as SCL:
   #IF_X3 := #X2 AND #aktr_GRFR AND NOT #snsr_KV;
END_REGION

REGION Network 9: Schritt 3 / Flip-Flop
   RUNG wire#powerrail
      Contact( #IF_X3 )
      S_SR(operand := #X3, r1 := #X4)
   END_RUNG
   // the same network as SCL:
   IF #IF_X3 THEN
       #X3 := TRUE;   // SR flip-flop
   END_IF;
   IF #X4 THEN #X3 := FALSE; END_IF;
END_REGION

REGION Network 10: Schritt 3 /Handeln
   RUNG wire#powerrail
      Contact( #X3 )
      P_Trig( #flk_X3 )
      wire#w1
      R_Coil( #aktr_Z )
   END_RUNG
   RUNG wire#w1
      R_Coil( #Zmove_ended )
   END_RUNG
   // the same network as SCL:
   #_w1 := #X3 AND NOT #flk_X3;   // rising edge
   #flk_X3 := #X3;
   IF #_w1 THEN
       #aktr_Z := FALSE;
       #Zmove_ended := FALSE;
   END_IF;
END_REGION

REGION Network 11: Schritt 4 / Mit OT rueberfahren
   RUNG wire#powerrail
      Contact( #X3 )
      Contact( #Zmove_ended )
      Coil( #IF_X4 )
   END_RUNG
   // the same network as SCL:
   #IF_X4 := #X3 AND #Zmove_ended;
END_REGION

REGION Network 12: Schritt 4 /Flip-Flop
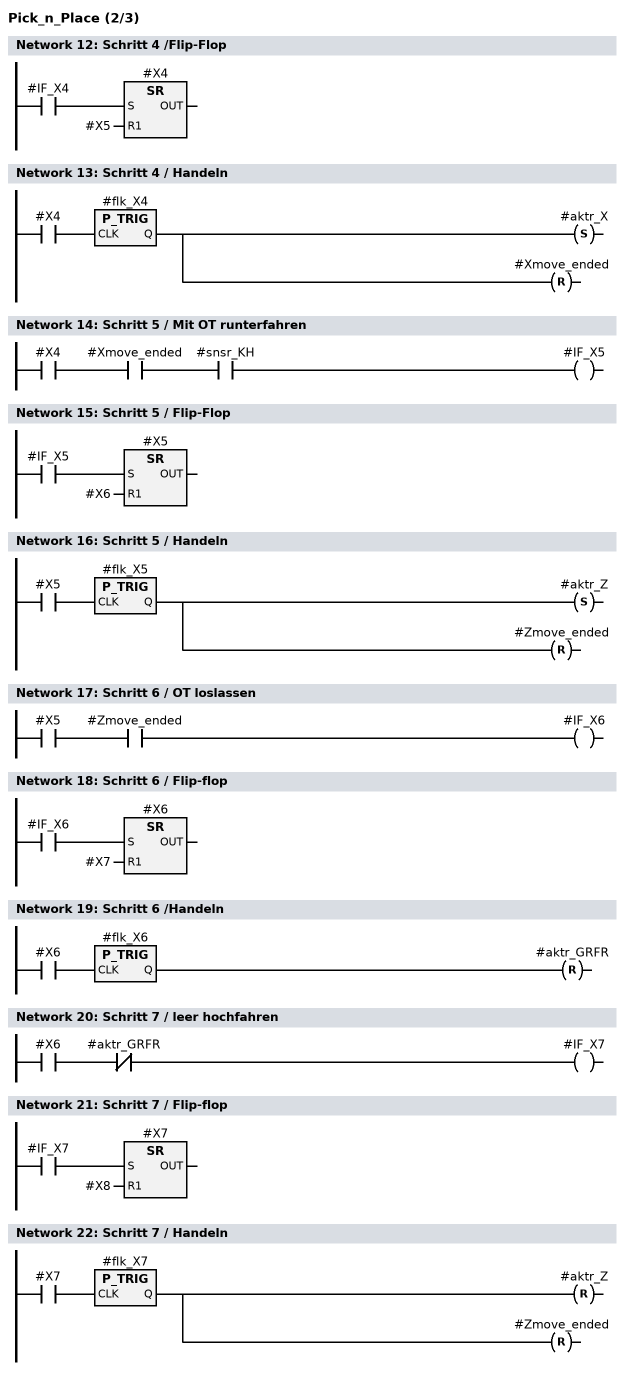
   RUNG wire#powerrail
      Contact( #IF_X4 )
      S_SR(operand := #X4, r1 := #X5)
   END_RUNG
   // the same network as SCL:
   IF #IF_X4 THEN
       #X4 := TRUE;   // SR flip-flop
   END_IF;
   IF #X5 THEN #X4 := FALSE; END_IF;
END_REGION

REGION Network 13: Schritt 4 / Handeln
   RUNG wire#powerrail
      Contact( #X4 )
      P_Trig( #flk_X4 )
      wire#w1
      S_Coil( #aktr_X )
   END_RUNG
   RUNG wire#w1
      R_Coil( #Xmove_ended )
   END_RUNG
   // the same network as SCL:
   #_w1 := #X4 AND NOT #flk_X4;   // rising edge
   #flk_X4 := #X4;
   IF #_w1 THEN
       #aktr_X := TRUE;
       #Xmove_ended := FALSE;
   END_IF;
END_REGION

REGION Network 14: Schritt 5 / Mit OT runterfahren
   RUNG wire#powerrail
      Contact( #X4 )
      Contact( #Xmove_ended )
      Contact( #snsr_KH )
      Coil( #IF_X5 )
   END_RUNG
   // the same network as SCL:
   #IF_X5 := #X4 AND #Xmove_ended AND #snsr_KH;
END_REGION

REGION Network 15: Schritt 5 / Flip-Flop
   RUNG wire#powerrail
      Contact( #IF_X5 )
      S_SR(operand := #X5, r1 := #X6)
   END_RUNG
   // the same network as SCL:
   IF #IF_X5 THEN
       #X5 := TRUE;   // SR flip-flop
   END_IF;
   IF #X6 THEN #X5 := FALSE; END_IF;
END_REGION

REGION Network 16: Schritt 5 / Handeln
   RUNG wire#powerrail
      Contact( #X5 )
      P_Trig( #flk_X5 )
      wire#w1
      S_Coil( #aktr_Z )
   END_RUNG
   RUNG wire#w1
      R_Coil( #Zmove_ended )
   END_RUNG
   // the same network as SCL:
   #_w1 := #X5 AND NOT #flk_X5;   // rising edge
   #flk_X5 := #X5;
   IF #_w1 THEN
       #aktr_Z := TRUE;
       #Zmove_ended := FALSE;
   END_IF;
END_REGION

REGION Network 17: Schritt 6 / OT loslassen
   RUNG wire#powerrail
      Contact( #X5 )
      Contact( #Zmove_ended )
      Coil( #IF_X6 )
   END_RUNG
   // the same network as SCL:
   #IF_X6 := #X5 AND #Zmove_ended;
END_REGION

REGION Network 18: Schritt 6 / Flip-flop
   RUNG wire#powerrail
      Contact( #IF_X6 )
      S_SR(operand := #X6, r1 := #X7)
   END_RUNG
   // the same network as SCL:
   IF #IF_X6 THEN
       #X6 := TRUE;   // SR flip-flop
   END_IF;
   IF #X7 THEN #X6 := FALSE; END_IF;
END_REGION

REGION Network 19: Schritt 6 /Handeln
   RUNG wire#powerrail
      Contact( #X6 )
      P_Trig( #flk_X6 )
      R_Coil( #aktr_GRFR )
   END_RUNG
   // the same network as SCL:
   #_w1 := #X6 AND NOT #flk_X6;   // rising edge
   #flk_X6 := #X6;
   IF #_w1 THEN #aktr_GRFR := FALSE; END_IF;
END_REGION

REGION Network 20: Schritt 7 / leer hochfahren
   RUNG wire#powerrail
      Contact( #X6 )
      I_Contact( #aktr_GRFR )
      Coil( #IF_X7 )
   END_RUNG
   // the same network as SCL:
   #IF_X7 := #X6 AND NOT #aktr_GRFR;
END_REGION

REGION Network 21: Schritt 7 / Flip-flop
   RUNG wire#powerrail
      Contact( #IF_X7 )
      S_SR(operand := #X7, r1 := #X8)
   END_RUNG
   // the same network as SCL:
   IF #IF_X7 THEN
       #X7 := TRUE;   // SR flip-flop
   END_IF;
   IF #X8 THEN #X7 := FALSE; END_IF;
END_REGION

REGION Network 22: Schritt 7 / Handeln
   RUNG wire#powerrail
      Contact( #X7 )
      P_Trig( #flk_X7 )
      wire#w1
      R_Coil( #aktr_Z )
   END_RUNG
   RUNG wire#w1
      R_Coil( #Zmove_ended )
   END_RUNG
   // the same network as SCL:
   #_w1 := #X7 AND NOT #flk_X7;   // rising edge
   #flk_X7 := #X7;
   IF #_w1 THEN
       #aktr_Z := FALSE;
       #Zmove_ended := FALSE;
   END_IF;
END_REGION

REGION Network 23: Schritt 8 / leer zur Grundstellung
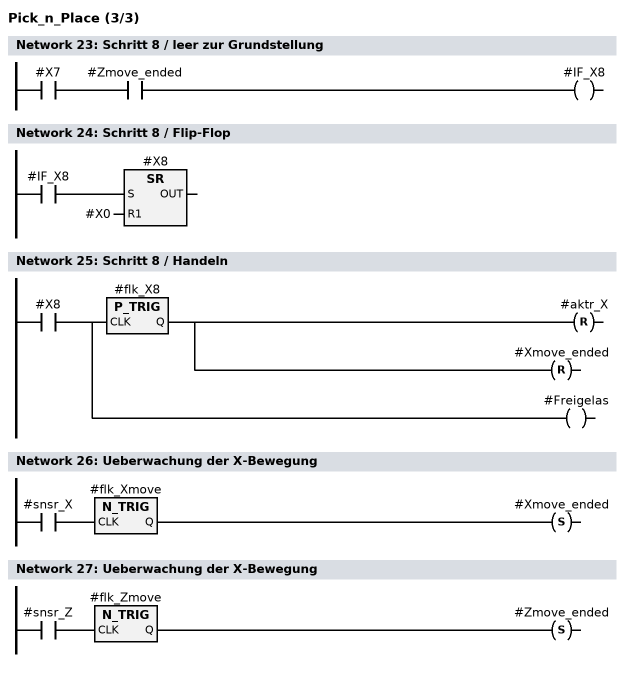
   RUNG wire#powerrail
      Contact( #X7 )
      Contact( #Zmove_ended )
      Coil( #IF_X8 )
   END_RUNG
   // the same network as SCL:
   #IF_X8 := #X7 AND #Zmove_ended;
END_REGION

REGION Network 24: Schritt 8 / Flip-Flop
   RUNG wire#powerrail
      Contact( #IF_X8 )
      S_SR(operand := #X8, r1 := #X0)
   END_RUNG
   // the same network as SCL:
   IF #IF_X8 THEN
       #X8 := TRUE;   // SR flip-flop
   END_IF;
   IF #X0 THEN #X8 := FALSE; END_IF;
END_REGION

REGION Network 25: Schritt 8 / Handeln
   RUNG wire#powerrail
      Contact( #X8 )
      wire#w1
      P_Trig( #flk_X8 )
      wire#w2
      R_Coil( #aktr_X )
   END_RUNG
   RUNG wire#w2
      R_Coil( #Xmove_ended )
   END_RUNG
   RUNG wire#w1
      Coil( #Freigelas )
   END_RUNG
   // the same network as SCL:
   #_w1 := #X8 AND NOT #flk_X8;   // rising edge
   #flk_X8 := #X8;
   IF #_w1 THEN
       #aktr_X := FALSE;
       #Xmove_ended := FALSE;
   END_IF;
   #Freigelas := #X8;
END_REGION

REGION Network 26: Ueberwachung der X-Bewegung
   RUNG wire#powerrail
      Contact( #snsr_X )
      N_Trig( #flk_Xmove )
      S_Coil( #Xmove_ended )
   END_RUNG
   // the same network as SCL:
   #_w1 := NOT #snsr_X AND #flk_Xmove;   // falling edge
   #flk_Xmove := #snsr_X;
   IF #_w1 THEN #Xmove_ended := TRUE; END_IF;
END_REGION

REGION Network 27: Ueberwachung der X-Bewegung
   RUNG wire#powerrail
      Contact( #snsr_Z )
      N_Trig( #flk_Zmove )
      S_Coil( #Zmove_ended )
   END_RUNG
   // the same network as SCL:
   #_w1 := NOT #snsr_Z AND #flk_Zmove;   // falling edge
   #flk_Zmove := #snsr_Z;
   IF #_w1 THEN #Zmove_ended := TRUE; END_IF;
END_REGION
END_FUNCTION_BLOCK

FUNCTION_BLOCK "03_02_Bearbeitungszelle"   // FB6, FBD
{ S7_Optimized_Access := 'FALSE' }
VERSION : 0.1
   VAR_INPUT
      Start : Bool;
      snsr_Eingang : Bool;
      snsr_V : Bool;
      snsr_H : Bool;
      Sperre : Bool;
      Freigabe_IN : Bool;
      Motor_An : Bool;
   END_VAR
   VAR_OUTPUT
      "aktr_OT/UT" : Bool;
      aktr_MTR : Bool;
   END_VAR
   VAR
      Teile_Typ : Bool;
      flk_snsr_Eingang : Bool;
      Beladen : Bool;
      flk_snsr_H : Bool;
      flk_P_sens_H : Bool;
   END_VAR
   VAR_TEMP   // added for the SCL form of the ladder/FBD networks
      _w1 : Bool;
   END_VAR
BEGIN

REGION Network 1: Stromstoß-Schalter für OT/UT
   // Wird abwächseld OT und UT hergestellt
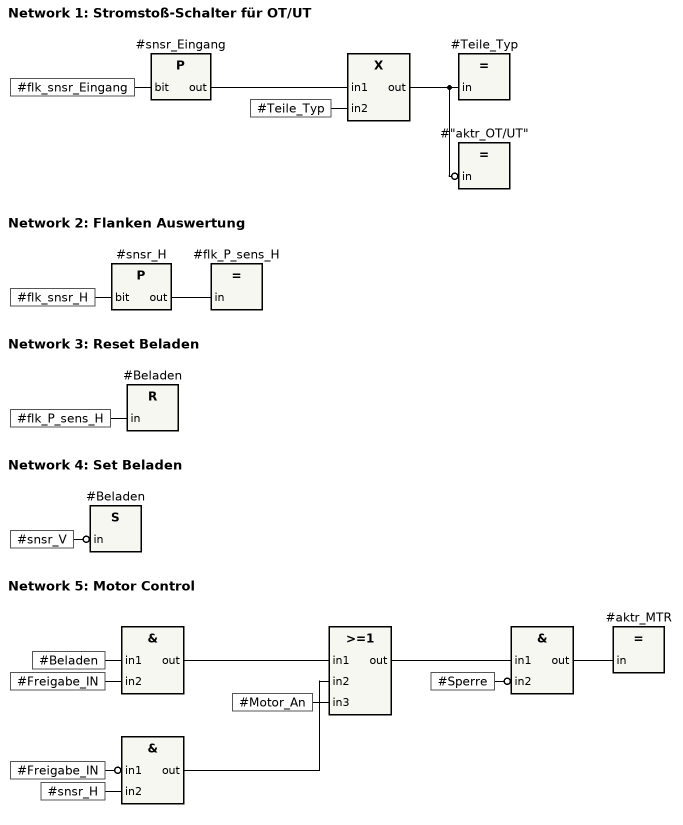
   #_w1 := #snsr_Eingang AND NOT #flk_snsr_Eingang;   // rising edge of #snsr_Eingang
   #flk_snsr_Eingang := #snsr_Eingang;
   #Teile_Typ := #_w1 XOR #Teile_Typ;
   #"aktr_OT/UT" := NOT #Teile_Typ;
END_REGION

REGION Network 2: Flanken Auswertung
   #_w1 := #snsr_H AND NOT #flk_snsr_H;   // rising edge of #snsr_H
   #flk_snsr_H := #snsr_H;
   #flk_P_sens_H := #_w1;
END_REGION

REGION Network 3: Reset Beladen
   // Reset des Statuses BELADEN des ersten Förderbandes
   IF #flk_P_sens_H THEN #Beladen := FALSE; END_IF;
END_REGION

REGION Network 4: Set Beladen
   // Set des Statuses BELADEN des ersten Förderbandes
   IF NOT #snsr_V THEN #Beladen := TRUE; END_IF;
END_REGION

REGION Network 5: Motor Control
   // Motorkontrolle der ersten Förderband
   #aktr_MTR := ((#Beladen AND #Freigabe_IN) OR (NOT #Freigabe_IN AND #snsr_H) OR #Motor_An) AND NOT #Sperre;
END_REGION
END_FUNCTION_BLOCK

FUNCTION_BLOCK "03_03_Weiche"   // FB7, LAD
{ S7_Optimized_Access := 'FALSE' }
VERSION : 0.1
   VAR_INPUT
      FRGB_IN_OT : Bool;
      FRGB_IN_UT : Bool;
      snsr_OT : Bool;
      snsr_UT : Bool;
      snsr_OT_V : Bool;
      snsr_OT_H : Bool;
      snsr_UT_V : Bool;
      snsr_UT_H : Bool;
      Sperre : Bool;
   END_VAR
   VAR_OUTPUT
      Freigabe_OUT : Bool;
      aktr_MTR_1_UT : Bool;
      aktr_MTR_2_UT : Bool;
      aktr_MTR_OT : Bool;
      aktr_SCHWNK_ARM : Bool;
      aktr_SCHWNK_BND : Bool;
      MTR_AN : Bool;
   END_VAR
   VAR
      Beladen_OT : Bool;
      Beladen_UT : Bool;
      flk_snsr_OT_V : Bool;
      flk_snsr_OT_H : Bool;
      flk_snsr_UT_V : Bool;
      flk_snsr_UT_H : Bool;
      flk_Aswertung : Bool;
      OT : Bool;
      UT : Bool;
      Delay : Time;
      IEC_TMR_0_INST : TP;
      flk_UT : Bool;
      flk_1_UT_H : Bool;
   END_VAR
   VAR_TEMP   // added for the SCL form of the ladder/FBD networks
      _w1 : Bool;
      _w2 : Bool;
   END_VAR
BEGIN

REGION Network 1: Flankenauswertung
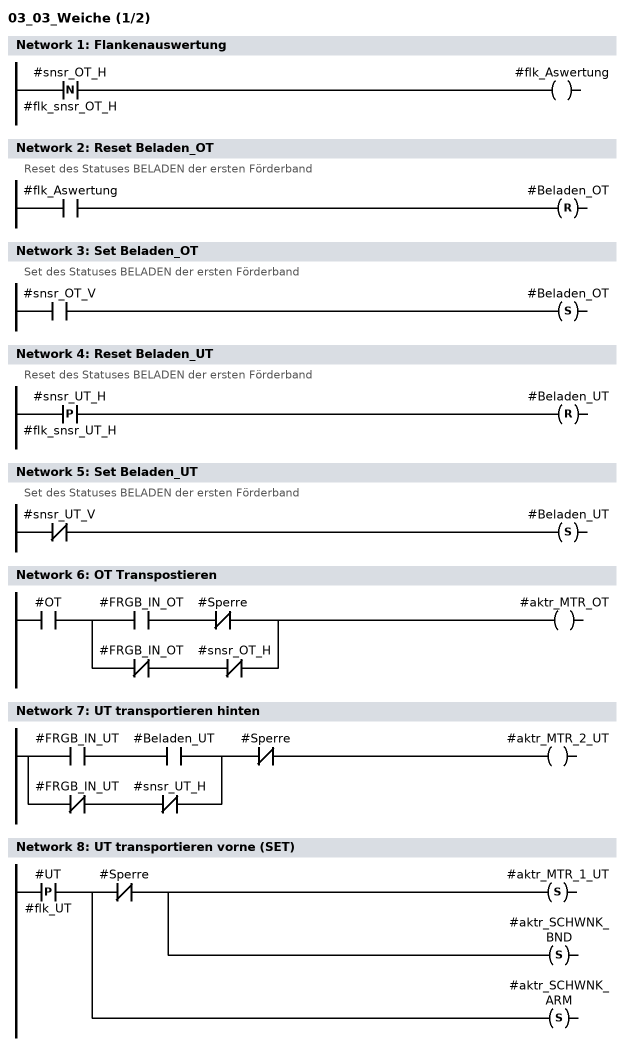
   RUNG wire#powerrail
      N_Contact(operand := #snsr_OT_H, bit := #flk_snsr_OT_H)
      Coil( #flk_Aswertung )
   END_RUNG
   // the same network as SCL:
   #_w1 := NOT #snsr_OT_H AND #flk_snsr_OT_H;   // falling edge of #snsr_OT_H
   #flk_snsr_OT_H := #snsr_OT_H;
   #flk_Aswertung := #_w1;
END_REGION

REGION Network 2: Reset Beladen_OT
   // Reset des Statuses BELADEN der ersten Förderband
   RUNG wire#powerrail
      Contact( #flk_Aswertung )
      R_Coil( #Beladen_OT )
   END_RUNG
   // the same network as SCL:
   IF #flk_Aswertung THEN #Beladen_OT := FALSE; END_IF;
END_REGION

REGION Network 3: Set Beladen_OT
   // Set des Statuses BELADEN der ersten Förderband
   RUNG wire#powerrail
      Contact( #snsr_OT_V )
      S_Coil( #Beladen_OT )
   END_RUNG
   // the same network as SCL:
   IF #snsr_OT_V THEN #Beladen_OT := TRUE; END_IF;
END_REGION

REGION Network 4: Reset Beladen_UT
   // Reset des Statuses BELADEN der ersten Förderband
   RUNG wire#powerrail
      P_Contact(operand := #snsr_UT_H, bit := #flk_snsr_UT_H)
      R_Coil( #Beladen_UT )
   END_RUNG
   // the same network as SCL:
   #_w1 := #snsr_UT_H AND NOT #flk_snsr_UT_H;   // rising edge of #snsr_UT_H
   #flk_snsr_UT_H := #snsr_UT_H;
   IF #_w1 THEN #Beladen_UT := FALSE; END_IF;
END_REGION

REGION Network 5: Set Beladen_UT
   // Set des Statuses BELADEN der ersten Förderband
   RUNG wire#powerrail
      I_Contact( #snsr_UT_V )
      S_Coil( #Beladen_UT )
   END_RUNG
   // the same network as SCL:
   IF NOT #snsr_UT_V THEN #Beladen_UT := TRUE; END_IF;
END_REGION

REGION Network 6: OT Transpostieren
   RUNG wire#powerrail
      Contact( #OT )
      wire#w1
      Contact( #FRGB_IN_OT )
      I_Contact( #Sperre )
      wire#w2
      Coil( #aktr_MTR_OT )
   END_RUNG
   RUNG wire#w1
      I_Contact( #FRGB_IN_OT )
      I_Contact( #snsr_OT_H )
   END_RUNG wire#w2
   // the same network as SCL:
   #aktr_MTR_OT := #OT AND ((#FRGB_IN_OT AND NOT #Sperre) OR (NOT #FRGB_IN_OT AND NOT #snsr_OT_H));
END_REGION

REGION Network 7: UT transportieren hinten
   RUNG wire#powerrail
      Contact( #FRGB_IN_UT )
      Contact( #Beladen_UT )
      wire#w1
      I_Contact( #Sperre )
      Coil( #aktr_MTR_2_UT )
   END_RUNG
   RUNG wire#powerrail
      I_Contact( #FRGB_IN_UT )
      I_Contact( #snsr_UT_H )
   END_RUNG wire#w1
   // the same network as SCL:
   #aktr_MTR_2_UT := ((#FRGB_IN_UT AND #Beladen_UT) OR (NOT #FRGB_IN_UT AND NOT #snsr_UT_H)) AND NOT #Sperre;
END_REGION

REGION Network 8: UT transportieren vorne (SET)
   RUNG wire#powerrail
      P_Contact(operand := #UT, bit := #flk_UT)
      wire#w1
      I_Contact( #Sperre )
      wire#w2
      S_Coil( #aktr_MTR_1_UT )
   END_RUNG
   RUNG wire#w2
      S_Coil( #aktr_SCHWNK_BND )
   END_RUNG
   RUNG wire#w1
      S_Coil( #aktr_SCHWNK_ARM )
   END_RUNG
   // the same network as SCL:
   #_w1 := #UT AND NOT #flk_UT;   // rising edge of #UT
   #flk_UT := #UT;
   IF #_w1 AND NOT #Sperre THEN
       #aktr_MTR_1_UT := TRUE;
       #aktr_SCHWNK_BND := TRUE;
   END_IF;
   IF #_w1 THEN #aktr_SCHWNK_ARM := TRUE; END_IF;
END_REGION

REGION Network 9: UT transportieren vorne (RESET)
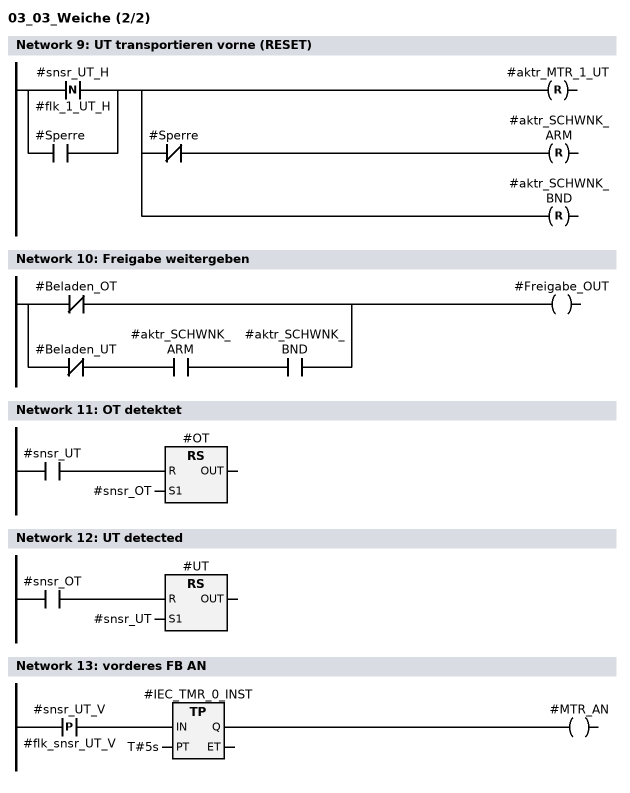
   RUNG wire#powerrail
      N_Contact(operand := #snsr_UT_H, bit := #flk_1_UT_H)
      wire#w1
      R_Coil( #aktr_MTR_1_UT )
   END_RUNG
   RUNG wire#powerrail
      Contact( #Sperre )
   END_RUNG wire#w1
   RUNG wire#w1
      I_Contact( #Sperre )
      R_Coil( #aktr_SCHWNK_ARM )
   END_RUNG
   RUNG wire#w1
      R_Coil( #aktr_SCHWNK_BND )
   END_RUNG
   // the same network as SCL:
   #_w1 := NOT #snsr_UT_H AND #flk_1_UT_H;   // falling edge of #snsr_UT_H
   #flk_1_UT_H := #snsr_UT_H;
   #_w2 := #_w1 OR #Sperre;
   IF #_w2 THEN #aktr_MTR_1_UT := FALSE; END_IF;
   IF #_w2 AND NOT #Sperre THEN #aktr_SCHWNK_ARM := FALSE; END_IF;
   IF #_w2 THEN #aktr_SCHWNK_BND := FALSE; END_IF;
END_REGION

REGION Network 10: Freigabe weitergeben
   RUNG wire#powerrail
      I_Contact( #Beladen_OT )
      wire#w1
      Coil( #Freigabe_OUT )
   END_RUNG
   RUNG wire#powerrail
      I_Contact( #Beladen_UT )
      Contact( #aktr_SCHWNK_ARM )
      Contact( #aktr_SCHWNK_BND )
   END_RUNG wire#w1
   // the same network as SCL:
   #Freigabe_OUT := NOT #Beladen_OT OR (NOT #Beladen_UT AND #aktr_SCHWNK_ARM AND #aktr_SCHWNK_BND);
END_REGION

REGION Network 11: OT detektet
   RUNG wire#powerrail
      Contact( #snsr_UT )
      S_RS(operand := #OT, s1 := #snsr_OT)
   END_RUNG
   // the same network as SCL:
   IF #snsr_UT THEN
       #OT := FALSE;   // RS flip-flop
   END_IF;
   IF #snsr_OT THEN #OT := TRUE; END_IF;
END_REGION

REGION Network 12: UT detected
   RUNG wire#powerrail
      Contact( #snsr_OT )
      S_RS(operand := #UT, s1 := #snsr_UT)
   END_RUNG
   // the same network as SCL:
   IF #snsr_OT THEN
       #UT := FALSE;   // RS flip-flop
   END_IF;
   IF #snsr_UT THEN #UT := TRUE; END_IF;
END_REGION

REGION Network 13: vorderes FB AN
   #_w1 := #snsr_UT_V AND NOT #flk_snsr_UT_V;   // rising edge of #snsr_UT_V
   #flk_snsr_UT_V := #snsr_UT_V;
   #IEC_TMR_0_INST.TP(IN := #_w1, PT := T#5s);
   #MTR_AN := #IEC_TMR_0_INST.Q;
END_REGION
END_FUNCTION_BLOCK

FUNCTION "Steuerung" : Void   // FC1, FBD
{ S7_Optimized_Access := 'FALSE' }
VERSION : 0.1
   VAR_TEMP   // added for the SCL form of the ladder/FBD networks
      _w1 : Bool;
   END_VAR
BEGIN

REGION Network 1: Not-Halt
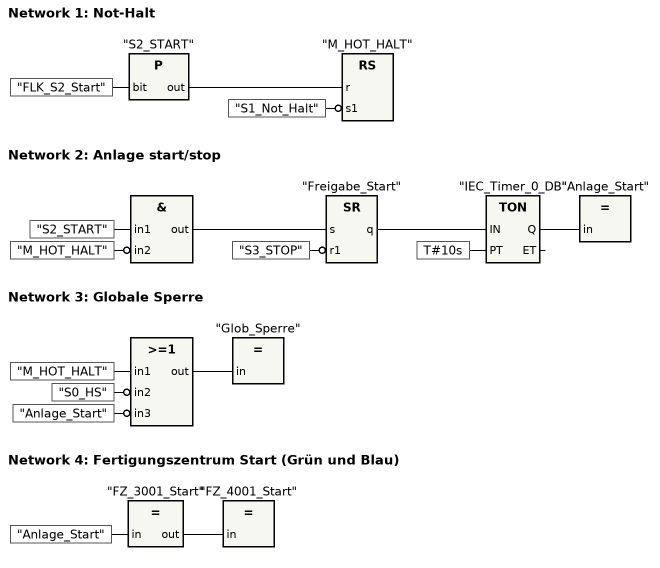
   #_w1 := "S2_START" AND NOT "FLK_S2_Start";   // rising edge of "S2_START"
   "FLK_S2_Start" := "S2_START";
   IF #_w1 THEN
       "M_HOT_HALT" := FALSE;   // RS flip-flop
   END_IF;
   IF NOT "S1_Not_Halt" THEN "M_HOT_HALT" := TRUE; END_IF;
END_REGION

REGION Network 2: Anlage start/stop
   IF "S2_START" AND NOT "M_HOT_HALT" THEN
       "Freigabe_Start" := TRUE;   // SR flip-flop
   END_IF;
   IF NOT "S3_STOP" THEN "Freigabe_Start" := FALSE; END_IF;
   "IEC_Timer_0_DB".TON(IN := "Freigabe_Start", PT := T#10s);
   "Anlage_Start" := "IEC_Timer_0_DB".Q;
END_REGION

REGION Network 3: Globale Sperre
   "Glob_Sperre" := "M_HOT_HALT" OR NOT "S0_HS" OR NOT "Anlage_Start";
END_REGION

REGION Network 4: Fertigungszentrum Start (Grün und Blau)
   "FZ_3001_Start" := "Anlage_Start";
   "FZ_4001_Start" := "Anlage_Start";
END_REGION
END_FUNCTION

FUNCTION "Output" : Void   // FC3, LAD
TITLE = Hier steuern wir die Ausgänge
{ S7_Optimized_Access := 'FALSE' }
VERSION : 0.1
   VAR_TEMP   // added for the SCL form of the ladder/FBD networks
      _w1 : Bool;
   END_VAR
BEGIN

REGION Network 1: Schaltkasten
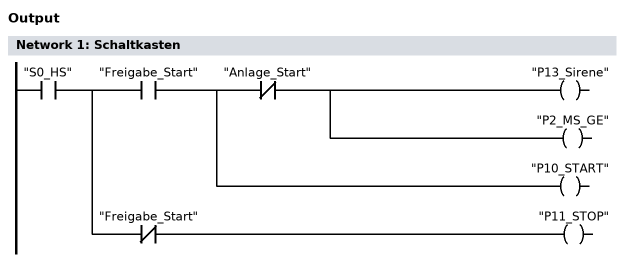
   RUNG wire#powerrail
      Contact( "S0_HS" )
      wire#w1
      Contact( "Freigabe_Start" )
      wire#w2
      I_Contact( "Anlage_Start" )
      wire#w3
      Coil( "P13_Sirene" )
   END_RUNG
   RUNG wire#w3
      Coil( "P2_MS_GE" )
   END_RUNG
   RUNG wire#w2
      Coil( "P10_START" )
   END_RUNG
   RUNG wire#w1
      I_Contact( "Freigabe_Start" )
      Coil( "P11_STOP" )
   END_RUNG
   // the same network as SCL:
   #_w1 := "S0_HS" AND "Freigabe_Start";
   "P13_Sirene" := #_w1 AND NOT "Anlage_Start";
   "P2_MS_GE" := "P13_Sirene";
   "P10_START" := #_w1;
   "P11_STOP" := "S0_HS" AND NOT "Freigabe_Start";
END_REGION
END_FUNCTION

ORGANIZATION_BLOCK "Main"   // OB1, FBD
TITLE = "Main Program Sweep (Cycle)"
{ S7_Optimized_Access := 'FALSE' }
VERSION : 0.1
   VAR_TEMP
      OB1_EV_CLASS : Byte;   // Bits 0-3 = 1 (Coming event), Bits 4-7 = 1 (Event class 1)
      OB1_SCAN_1 : Byte;   // 1 (Cold restart scan 1 of OB 1), 3 (Scan 2-n of OB 1)
      OB1_PRIORITY : Byte;   // Priority of OB Execution
      OB1_OB_NUMBR : Byte;   // 1 (Organization block 1, OB1)
      OB1_RESERVED_1 : Byte;   // Reserved for system
      OB1_RESERVED_2 : Byte;   // Reserved for system
      OB1_PREV_CYCLE : Int;   // Cycle time of previous OB1 scan (milliseconds)
      OB1_MIN_CYCLE : Int;   // Minimum cycle time of OB1 (milliseconds)
      OB1_MAX_CYCLE : Int;   // Maximum cycle time of OB1 (milliseconds)
      OB1_DATE_TIME : Date_And_Time;   // Date and time OB1 started
   END_VAR
BEGIN

REGION Network 1: Steuerung
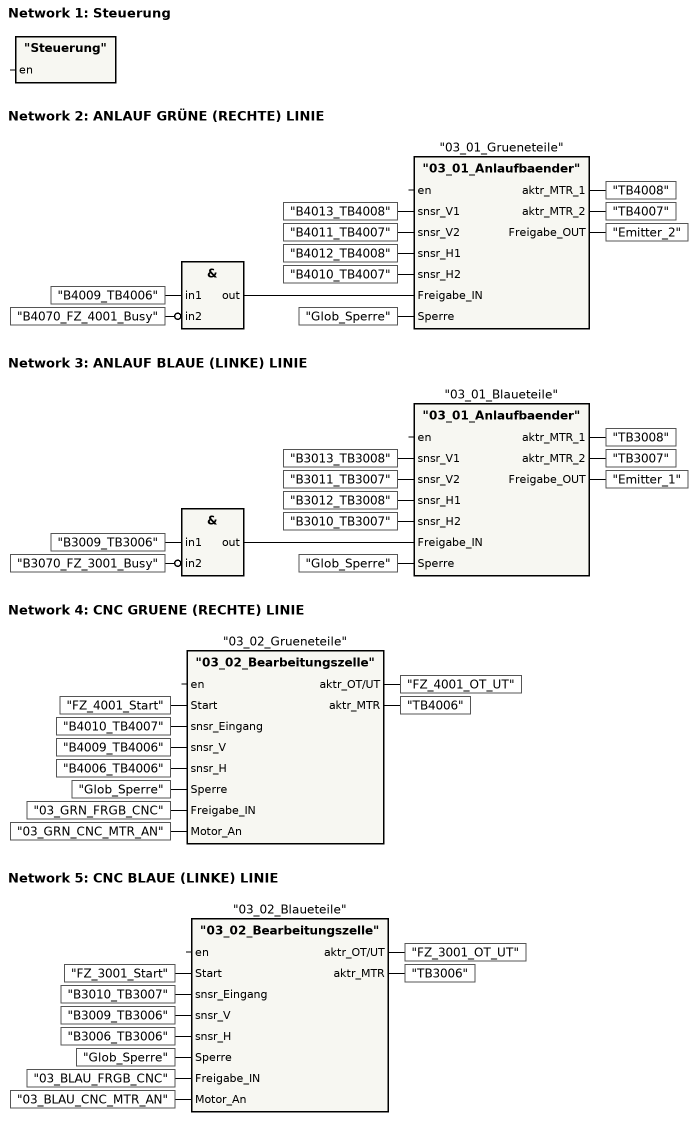
   "Steuerung"();
END_REGION

REGION Network 2: ANLAUF GRÜNE (RECHTE) LINIE
   "03_01_Grueneteile"(snsr_V1 := "B4013_TB4008",   // "03_01_Anlaufbaender"
                       snsr_V2 := "B4011_TB4007",
                       snsr_H1 := "B4012_TB4008",
                       snsr_H2 := "B4010_TB4007",
                       Freigabe_IN := "B4009_TB4006" AND NOT "B4070_FZ_4001_Busy",
                       Sperre := "Glob_Sperre",
                       aktr_MTR_1 => "TB4008",
                       aktr_MTR_2 => "TB4007",
                       Freigabe_OUT => "Emitter_2");
END_REGION

REGION Network 3: ANLAUF BLAUE (LINKE) LINIE
   "03_01_Blaueteile"(snsr_V1 := "B3013_TB3008",   // "03_01_Anlaufbaender"
                      snsr_V2 := "B3011_TB3007",
                      snsr_H1 := "B3012_TB3008",
                      snsr_H2 := "B3010_TB3007",
                      Freigabe_IN := "B3009_TB3006" AND NOT "B3070_FZ_3001_Busy",
                      Sperre := "Glob_Sperre",
                      aktr_MTR_1 => "TB3008",
                      aktr_MTR_2 => "TB3007",
                      Freigabe_OUT => "Emitter_1");
END_REGION

REGION Network 4: CNC GRUENE (RECHTE) LINIE
   "03_02_Grueneteile"(Start := "FZ_4001_Start",   // "03_02_Bearbeitungszelle"
                       snsr_Eingang := "B4010_TB4007",
                       snsr_V := "B4009_TB4006",
                       snsr_H := "B4006_TB4006",
                       Sperre := "Glob_Sperre",
                       Freigabe_IN := "03_GRN_FRGB_CNC",
                       Motor_An := "03_GRN_CNC_MTR_AN",
                       "aktr_OT/UT" => "FZ_4001_OT_UT",
                       aktr_MTR => "TB4006");
END_REGION

REGION Network 5: CNC BLAUE (LINKE) LINIE
   "03_02_Blaueteile"(Start := "FZ_3001_Start",   // "03_02_Bearbeitungszelle"
                      snsr_Eingang := "B3010_TB3007",
                      snsr_V := "B3009_TB3006",
                      snsr_H := "B3006_TB3006",
                      Sperre := "Glob_Sperre",
                      Freigabe_IN := "03_BLAU_FRGB_CNC",
                      Motor_An := "03_BLAU_CNC_MTR_AN",
                      "aktr_OT/UT" => "FZ_3001_OT_UT",
                      aktr_MTR => "TB3006");
END_REGION

REGION Network 6: WEICHE GRUENE (RECHTE) LINIE
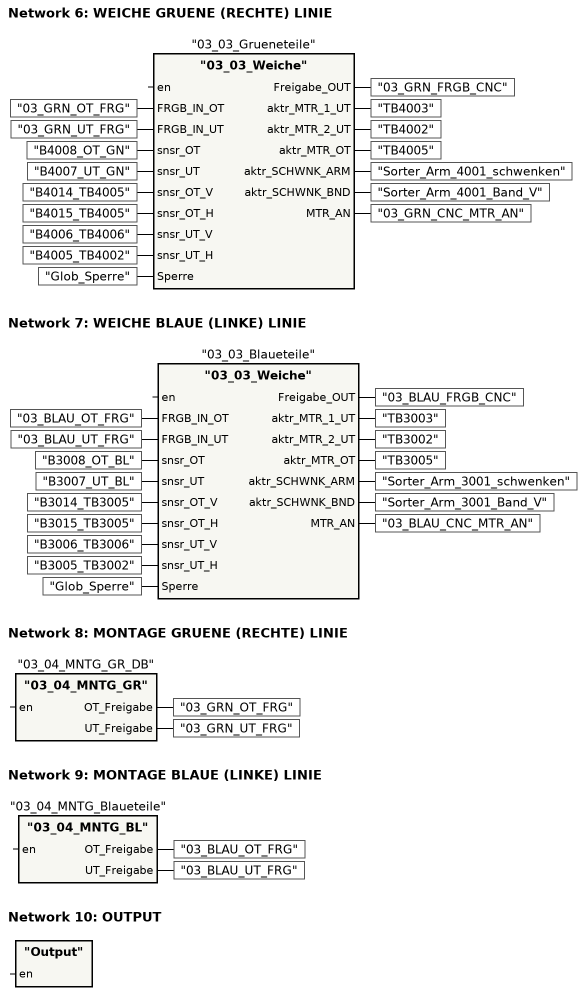
   "03_03_Grueneteile"(FRGB_IN_OT := "03_GRN_OT_FRG",   // "03_03_Weiche"
                       FRGB_IN_UT := "03_GRN_UT_FRG",
                       snsr_OT := "B4008_OT_GN",
                       snsr_UT := "B4007_UT_GN",
                       snsr_OT_V := "B4014_TB4005",
                       snsr_OT_H := "B4015_TB4005",
                       snsr_UT_V := "B4006_TB4006",
                       snsr_UT_H := "B4005_TB4002",
                       Sperre := "Glob_Sperre",
                       Freigabe_OUT => "03_GRN_FRGB_CNC",
                       aktr_MTR_1_UT => "TB4003",
                       aktr_MTR_2_UT => "TB4002",
                       aktr_MTR_OT => "TB4005",
                       aktr_SCHWNK_ARM => "Sorter_Arm_4001_schwenken",
                       aktr_SCHWNK_BND => "Sorter_Arm_4001_Band_V",
                       MTR_AN => "03_GRN_CNC_MTR_AN");
END_REGION

REGION Network 7: WEICHE BLAUE (LINKE) LINIE
   "03_03_Blaueteile"(FRGB_IN_OT := "03_BLAU_OT_FRG",   // "03_03_Weiche"
                      FRGB_IN_UT := "03_BLAU_UT_FRG",
                      snsr_OT := "B3008_OT_BL",
                      snsr_UT := "B3007_UT_BL",
                      snsr_OT_V := "B3014_TB3005",
                      snsr_OT_H := "B3015_TB3005",
                      snsr_UT_V := "B3006_TB3006",
                      snsr_UT_H := "B3005_TB3002",
                      Sperre := "Glob_Sperre",
                      Freigabe_OUT => "03_BLAU_FRGB_CNC",
                      aktr_MTR_1_UT => "TB3003",
                      aktr_MTR_2_UT => "TB3002",
                      aktr_MTR_OT => "TB3005",
                      aktr_SCHWNK_ARM => "Sorter_Arm_3001_schwenken",
                      aktr_SCHWNK_BND => "Sorter_Arm_3001_Band_V",
                      MTR_AN => "03_BLAU_CNC_MTR_AN");
END_REGION

REGION Network 8: MONTAGE GRUENE (RECHTE) LINIE
   "03_04_MNTG_GR_DB"(OT_Freigabe => "03_GRN_OT_FRG", UT_Freigabe => "03_GRN_UT_FRG");   // "03_04_MNTG_GR"
END_REGION

REGION Network 9: MONTAGE BLAUE (LINKE) LINIE
   "03_04_MNTG_Blaueteile"(OT_Freigabe => "03_BLAU_OT_FRG", UT_Freigabe => "03_BLAU_UT_FRG");   // "03_04_MNTG_BL"
END_REGION

REGION Network 10: OUTPUT
   "Output"();
END_REGION
END_ORGANIZATION_BLOCK

// ===== library: MasterCopy "RB_TB_einfach" =====

FUNCTION_BLOCK "RB_TB_einfach"   // FB101, GRAPH
{ S7_Optimized_Access := 'FALSE' }
VERSION : 0.1
// Einfacher Steuerbaustein RB / TB 
// Sensor Anfang / Ende  NO
   VAR_INPUT
      INIT_SQ : Bool := false;   // Kette in Initialzustand versetzen
      A_EIN : Bool;
      A_NOT_HALT : Bool;
      Nachfolgendes_Agg_frei : Bool;
      Sensor_vorheriges_Agg : Bool;
      Sensor_Anfang : Bool;   // Öffner
      Sensor_Ende : Bool;   // Öffner
   END_VAR
   VAR_OUTPUT
      Schritt_Nummer : Int;
      Aggregat : Bool;
      Aggregat_frei : Bool;
   END_VAR
   VAR
      HM_FLAM : Array[1..8] of Bool;
      Flanke : Array[1..8] of Bool;
      HM_Agg_Frei : Bool;
      HM_belegt : Bool;
      SWITCH : Array[0..0] of DWord;
      SW_SQTS : Array[0..6] of Byte;
      SW_ADDR : Word := 16#C;
      G7T_0 : GraphTransition;
      G7S_0 : GraphStep;
      PRE_CRIT : Array[0..1] of DWord;
      POST_CRIT : Array[0..0] of DWord;
      TVX : Array[0..2] of Byte;
      TTX : Array[0..2] of Byte;
      TSX : Array[0..2] of Byte;
      S00X : Array[0..2] of Byte;
      SOFFX : Array[0..2] of Byte;
      SONX : Array[0..2] of Byte;
      SAX : Array[0..2] of Byte;
      SERRX : Array[0..7] of Byte;
      SMX : Array[0..7] of Byte;
      S0X : Array[0..7] of Byte;
      S1X : Array[0..7] of Byte;
      S_DISPLAY : Int;   // Interne Anzeige des Ausgangsparameters S_NO
      S_SEL_OLD : Int;   // Vorheriger Wert an S_SEL
      S_DISPIDX : Byte;   // Index des Schritts, der an S_NO anliegt
      T_DISPIDX : Byte;   // Index der Transition, die an T_NO anliegt
      MOPEDGE : Struct
         AUTO : Bool := false;
         MAN : Bool := false;
         TAP : Bool := false;
         TOP : Bool := false;
         ACK_S : Bool := false;
         REG_S : Bool := false;
         T_PREV : Bool := false;
         T_NEXT : Bool := false;
         LOCK : Bool := false;
         SUP : Bool := false;
         ACKREQ : Bool := false;
         SSKIP : Bool := false;
         OFF : Bool := false;
         INIT : Bool := false;
         HALT : Bool := false;
         TMS_HALT : Bool := false;
         OPS_ZERO : Bool := false;
         SACT_DISP : Bool := false;
         SEF_DISP : Bool := false;
         SALL_DISP : Bool := false;
         S_PREV : Bool := false;
         S_NEXT : Bool := false;
         S_SELOK : Bool := false;
         S_ON : Bool := false;
         S_OFF : Bool := false;
         T_PUSH : Bool := false;
         REG : Bool := false;
         ACK : Bool := false;
         IL_PERM : Bool := false;
         T_PERM : Bool := false;
         ILP_MAN : Bool := false;
      END_STRUCT;
      MOP : Struct   // Betriebsart
         AUTO : Bool := true;   // Zustand: Automatischer Betrieb
         MAN : Bool := false;   // Zustand: Handbetrieb
         TAP : Bool := false;   // Zustand: Halbautomatisch/Weiterschalten mit Transition
         TOP : Bool := false;   // Zustand: Halbautomatisch/Ignoriere Transition
         ACK_S : Bool := false;   // Anforderung: Schritt quittieren, der an Parameter S_NO anliegt
         REG_S : Bool := false;   // Anforderung: Schritt registrieren, der an Parameter S_NO anliegt
         T_PREV : Bool := false;   // Anforderung: Vorherige gültige Transition am Parameter T_NO ausgeben
         T_NEXT : Bool := false;   // Anforderung: Nächste gültige Transition am Parameter T_NO ausgeben
         LOCK : Bool := true;   // Zustand: Interlockbearbeitung aktiviert
         SUP : Bool := true;   // Zustand: Supervisionsbearbeitung aktiviert
         ACKREQ : Bool := false;   // Zustand: Quittierung erforderlich
         SSKIP : Bool := false;   // Zustand: "Schritte überspringen" aktiviert
         OFF : Bool := false;   // Anforderung: Alle Schritte deaktivieren
         INIT : Bool := true;   // Anforderung: Kette in Initialzustand schalten
         HALT : Bool := false;   // Zustand: Kette schaltet nicht weiter
         TMS_HALT : Bool := false;   // Zustand: Alle internen Zeiten angehalten
         OPS_ZERO : Bool := false;   // Zustand: Alle mit N, L, D bearbeitete Operanden auf 0 gesetzt
         SACT_DISP : Bool := true;   // Zustand: Nur aktive Schritte anzeigen
         SEF_DISP : Bool := false;   // Zustand: Nur fehlerhafte und gestörte Schritte anzeigen
         SALL_DISP : Bool := false;   // Zustand: Alle Schritte anzeigen
         S_PREV : Bool := false;   // Anforderung: Vorherigen Schritt am Parameter S_NO ausgeben
         S_NEXT : Bool := false;   // Anforderung: Nächsten Schritt am Parameter S_NO ausgeben
         S_SELOK : Bool := false;   // Anforderung: Schrittnummer, die am Parameter S_SEL anliegt, am Parameter S_NO ausgeben
         S_ON : Bool := false;   // Anforderung: Schritt aktivieren, der am Parameter S_NO anliegt
         S_OFF : Bool := false;   // Anforderung: Schritt deaktivieren, der am Parameter S_NO anliegt
         T_PUSH : Bool := false;   // Anforderung: Schaltfreigabe für Transition
         REG : Bool := false;   // Anforderung: Alle Interlock- und Supervisionsfehler registrieren
         ACK : Bool := false;   // Anforderung: Alle Interlock- und Supervisionsfehler quittieren
         IL_PERM : Bool := false;   // Zustand: Permanente Bearbeitung aller Interlocks
         T_PERM : Bool := false;   // Zustand: Permanente Bearbeitung aller Transitionen
         ILP_MAN : Bool := false;   // Zustand: Permanente Bearbeitung aller Interlocks im Handbetrieb
      END_STRUCT;
      TICKS : Struct   // Zeittakte
         DELTA : Time := T#0ms;   // Zeitdifferenz zwischen zwei Zyklen
         OLD : Time := T#0ms;   // 10 ms Taktzählerstand im letzten Zyklus
         NEW : Time := T#0ms;   // 10 ms Taktzählerstand in diesem Zyklus
      END_STRUCT;
      SQ_FLAGS : Struct   // Kettenmerker
         ERR_FLT : Bool := false;   // Sammelfehler Interlock und Supervision
         ERROR : Bool := false;   // Sammelfehler Interlock
         FAULT : Bool := false;   // Sammelfehler Supervision
         RT_FAIL : Bool := false;   // Laufzeitfehler
         NO_SNO : Bool := false;   // Angeforderte Schrittnummer nicht gefunden
         NF_OFL : Bool := false;   // Überlauf: Zu viele Anforderungen ON oder OFF
         SA_OFL : Bool := false;   // Überlauf: Zu viele Schritte aktiv
         TV_OFL : Bool := false;   // Überlauf: Zu viele gültige Transitionen
         MSG_OFL : Bool := false;   // Überlauf: Nicht genügend Systemressourcen fü ALARM_S
         NO_SWI : Bool := false;   // Nicht Schalten in diesem Zyklus
         CYC_OP : Bool := false;   // Zyklische Bearbeitung der Kette nach Initialisierung
         AS_MSG : Bool := true;   // Meldungen zur Laufzeit durch Anweisung aktiviert oder deaktiviert
         AS_SEND : Bool := false;   // Meldungen von WR_USMSG senden oder nur in Diagnosepuffer eintragen
         SQ_BUSY : Bool := false;   // Interner Flankenmerker für Vorgangsbearbeitung
         SA_BUSY : Bool := false;   // Interner Flankenmerker für Vorgangsbearbeitung
         AS_SIG : Bool := false;   // Flankenmerker für Meldungen von Alarm_S und Alarm_SQ
      END_STRUCT;
      S_PTR : DWord := 16#450;
      S_PTR2 : DWord := 16#0;
      S_PTR3 : DWord := 16#D50;
      S_PTR4 : DWord := 16#D10;
      T_PTR : DWord := 16#CD0;
      C_AR2 : DWord := 16#0;
      M_FBDB : DWord := 16#640000;
      M_SNO : Word := 16#4;
      M_EVID : Word := 16#0;
      M_EVIL : C_Alarm_s;
      M_EVSV : C_Alarm_s;
      M_EV : DWord := 16#C30;
      CRIT : Array[0..31] of Bool;
      S_START : Byte := 16#0;
      S_IDX : Byte := 16#0;
      S_INT : Int := 72;
      S_TMP : Byte := 16#0;
      T_START : Byte := 16#0;
      T_IDX : Byte := 16#0;
      T_TMP : Byte := 16#0;
      T_TMP2 : Byte := 16#00;
      TV_POT : Byte := 16#02;
      RETURN1 : Byte := 16#0;
      RETURN2 : Byte := 16#0;
      SINI : Array[0..2] of Byte;
      LSTT : Array[0..6] of Byte;
      ATAJ : Array[0..6] of Byte;
      ATAB : Array[0..6] of Byte;
      PSTT : Array[0..6] of Byte;
      NSTT : Array[0..6] of Byte;
      ASSJ : Array[0..6] of Byte;
      ASSB : Array[0..6] of Byte;
      PTTS : Array[0..6] of Byte;
      NTTS : Array[0..6] of Byte;
      PRE_CNT : Word := 16#2;
      POST_CNT : Word := 16#1;
      ADR_COND : Word := 16#0;
      MAX_TVAL : Byte := 16#1;
      MAX_SACT : Byte := 16#1;
      MAX_CRIT : Byte := 16#4;
      T_CNT : Byte := 16#6;
      SUP_CNT : Byte := 16#0;
      LOCK_CNT : Byte := 16#5;
      S_CNT : Byte := 16#6;
      SQ_CNT : Byte := 16#1;
      PRS_INPAR : DWord := 16#40000000;
      PRS_OUTPAR : DWord := 16#0;
      GC_FLAGS : Struct
         T_MACH : Byte := 16#EB;
         COND_ED : Byte := 16#E2;
         W_LEVEL : Byte := 16#D5;
         FB_IF : Byte := 16#FA;
         AS_MSG : Word := 16#404;
         SSB : Word := 16#108;
         DILG : Word := 16#27E;
         ADDR_T0 : Word := 16#1A;
         CRIT_AVAIL : Bool := false;
         SSKIP_AVAIL : Bool := true;
         SSKIP_ON : Bool := false;
         ACK_REQ : Bool := false;
         SYNC_AVAIL : Bool := true;
         ILP_MAN : Bool := false;
         SWM_LOCKED : Bool := false;
         SAVE_SW : Bool := true;
      END_STRUCT;
      G7_FBMARK : Byte := 16#3C;
      G7_RELEASE : Byte := 16#3C;
      G7_ID2 : Byte := 16#37;
      G7_ID1 : Byte := 16#47;
   END_VAR
   // SW_SQTS[0] := 16#1;
   // TVX[0] := 16#1;
   // TTX[0] := 16#1;
   // TSX[0] := 16#1;
   // S00X[0] := 16#1;
   // SOFFX[0] := 16#1;
   // SONX[0] := 16#1;
   // SAX[0] := 16#1;
   // SERRX[0] := 16#1;
   // SMX[0] := 16#1;
   // S0X[0] := 16#1;
   // S1X[0] := 16#1;
   // SINI[0] := 16#2;
   // SINI[1] := 16#1;
   // SINI[2] := 0;
   // LSTT[0] := 0;
   // LSTT[1] := 0;
   // LSTT[2] := 0;
   // LSTT[3] := 0;
   // LSTT[4] := 0;
   // LSTT[5] := 0;
   // ATAJ[0] := 0;
   // ATAJ[1] := 16#1;
   // ATAJ[2] := 16#2;
   // ATAJ[3] := 16#3;
   // ATAJ[4] := 16#4;
   // ATAJ[5] := 16#5;
   // ATAB[0] := 0;
   // ATAB[1] := 16#1;
   // ATAB[2] := 16#2;
   // ATAB[3] := 16#3;
   // ATAB[4] := 16#4;
   // ATAB[5] := 16#5;
   // PSTT[0] := 0;
   // PSTT[1] := 16#1;
   // PSTT[2] := 16#2;
   // PSTT[3] := 16#3;
   // PSTT[4] := 16#4;
   // PSTT[5] := 16#5;
   // NSTT[0] := 16#1;
   // NSTT[1] := 16#2;
   // NSTT[2] := 16#3;
   // NSTT[3] := 16#4;
   // NSTT[4] := 16#5;
   // NSTT[5] := 16#6;
   // ASSJ[0] := 0;
   // ASSJ[1] := 16#1;
   // ASSJ[2] := 16#2;
   // ASSJ[3] := 16#3;
   // ASSJ[4] := 16#4;
   // ASSJ[5] := 16#5;
   // ASSB[0] := 0;
   // ASSB[1] := 16#1;
   // ASSB[2] := 16#2;
   // ASSB[3] := 16#3;
   // ASSB[4] := 16#4;
   // ASSB[5] := 16#5;
   // PTTS[0] := 0;
   // PTTS[2] := 16#1;
   // PTTS[3] := 16#2;
   // PTTS[4] := 16#3;
   // PTTS[5] := 16#4;
   // NTTS[0] := 0;
   // NTTS[1] := 16#1;
   // NTTS[2] := 16#2;
   // NTTS[3] := 16#3;
   // NTTS[4] := 16#4;
   // NTTS[5] := 16#5;
   // LSTT[6] := 16#1;
   // ATAJ[6] := 16#6;
   // ATAB[6] := 16#6;
   // PSTT[6] := 16#6;
   // NSTT[6] := 16#1;
   // ASSJ[6] := 16#6;
   // ASSB[6] := 16#6;
   // PTTS[6] := 16#5;
   // NTTS[6] := 16#6;
BEGIN
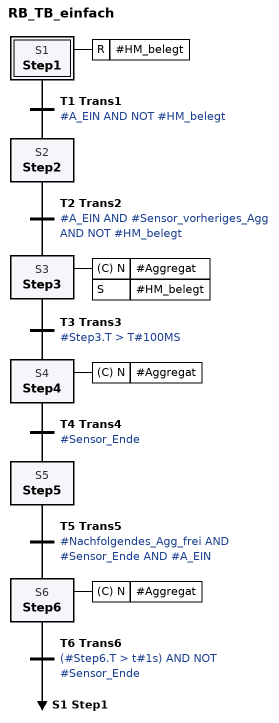
   // permanent pre-instructions
   NETWORK 1
      #HM_Agg_Frei := NOT #HM_belegt;
      #Aggregat_frei := NOT #HM_belegt;
   NETWORK 2
   TITLE = Ausgabe Schrittnummer
      #Schritt_Nummer := #S_DISPLAY;

   // sequencer 1
   INITIAL_STEP Step1:   // S1
      interlock C := NOT #A_NOT_HALT;
      // Warten auf Start
              R    #HM_belegt
   END_STEP
   TRANSITION Trans1 FROM Step1 TO Step2   // T1
      := #A_EIN AND NOT #HM_belegt;
   END_TRANSITION
   STEP Step4:   // S4
      interlock C := NOT #A_NOT_HALT;
      // Einfahrt bis Ende
      (C)     N    #Aggregat
   END_STEP
   TRANSITION Trans4 FROM Step4 TO Step5   // T4
      := #Sensor_Ende;
   END_TRANSITION
   STEP Step5:   // S5
      interlock C := NOT #A_NOT_HALT;
      // Warten auf Ausfahrt
   END_STEP
   TRANSITION Trans5 FROM Step5 TO Step6   // T5
      := #Nachfolgendes_Agg_frei AND #Sensor_Ende AND #A_EIN;
   END_TRANSITION
   STEP Step6:   // S6
      interlock C := NOT #A_NOT_HALT;
      // Ausfahrt bis Ende
      (C)     N    #Aggregat
   END_STEP
   TRANSITION Trans6 FROM Step6 TO Step1   // T6, jump
      := (#Step6.T > t#1s) AND NOT #Sensor_Ende;
   END_TRANSITION
   STEP Step3:   // S3
      interlock C := NOT #A_NOT_HALT;
      // Einfahrt Start
      (C)     N    #Aggregat
              S    #HM_belegt
   END_STEP
   TRANSITION Trans3 FROM Step3 TO Step4   // T3
      := #Step3.T > T#100MS;
   END_TRANSITION
   STEP Step2:   // S2
   END_STEP
   TRANSITION Trans2 FROM Step2 TO Step3   // T2
      := #A_EIN AND #Sensor_vorheriges_Agg AND NOT #HM_belegt;
   END_TRANSITION
END_FUNCTION_BLOCK

// ===== library: MasterCopy "Baustein_1" =====

FUNCTION_BLOCK "Baustein_1"   // FB2222, GRAPH
{ S7_Optimized_Access := 'FALSE' }
VERSION : 0.1
   VAR_INPUT
      INIT_SQ : Bool := false;   // Kette in Initialzustand versetzen
      A_EIN : Bool;
      A_NOT_HALT : Bool;
      Nachfolgendes_Agg_frei : Bool;
      Sensor_vorheriges_Agg : Bool;
      Sensor_Anfang : Bool;   // Öffner
      Sensor_Ende : Bool;   // Öffner
   END_VAR
   VAR_OUTPUT
      Schritt_Nummer : Int;
      Aggregat : Bool;
      Aggregat_frei : Bool;
   END_VAR
   VAR
      HM_FLAM : Array[1..8] of Bool;
      Flanke : Array[1..8] of Bool;
      HM_Agg_Frei : Bool;
      HM_belegt : Bool;
      SWITCH : Array[0..0] of DWord;
      SW_SQTS : Array[0..6] of Byte;
      SW_ADDR : Word := 16#C;
      G7T_0 : GraphTransition;
      G7S_0 : GraphStep;
      PRE_CRIT : Array[0..1] of DWord;
      POST_CRIT : Array[0..0] of DWord;
      TVX : Array[0..2] of Byte;
      TTX : Array[0..2] of Byte;
      TSX : Array[0..2] of Byte;
      S00X : Array[0..2] of Byte;
      SOFFX : Array[0..2] of Byte;
      SONX : Array[0..2] of Byte;
      SAX : Array[0..2] of Byte;
      SERRX : Array[0..7] of Byte;
      SMX : Array[0..7] of Byte;
      S0X : Array[0..7] of Byte;
      S1X : Array[0..7] of Byte;
      S_DISPLAY : Int;   // Interne Anzeige des Ausgangsparameters S_NO
      S_SEL_OLD : Int;   // Vorheriger Wert an S_SEL
      S_DISPIDX : Byte;   // Index des Schritts, der an S_NO anliegt
      T_DISPIDX : Byte;   // Index der Transition, die an T_NO anliegt
      MOPEDGE : Struct
         AUTO : Bool := false;
         MAN : Bool := false;
         TAP : Bool := false;
         TOP : Bool := false;
         ACK_S : Bool := false;
         REG_S : Bool := false;
         T_PREV : Bool := false;
         T_NEXT : Bool := false;
         LOCK : Bool := false;
         SUP : Bool := false;
         ACKREQ : Bool := false;
         SSKIP : Bool := false;
         OFF : Bool := false;
         INIT : Bool := false;
         HALT : Bool := false;
         TMS_HALT : Bool := false;
         OPS_ZERO : Bool := false;
         SACT_DISP : Bool := false;
         SEF_DISP : Bool := false;
         SALL_DISP : Bool := false;
         S_PREV : Bool := false;
         S_NEXT : Bool := false;
         S_SELOK : Bool := false;
         S_ON : Bool := false;
         S_OFF : Bool := false;
         T_PUSH : Bool := false;
         REG : Bool := false;
         ACK : Bool := false;
         IL_PERM : Bool := false;
         T_PERM : Bool := false;
         ILP_MAN : Bool := false;
      END_STRUCT;
      MOP : Struct   // Betriebsart
         AUTO : Bool := true;   // Zustand: Automatischer Betrieb
         MAN : Bool := false;   // Zustand: Handbetrieb
         TAP : Bool := false;   // Zustand: Halbautomatisch/Weiterschalten mit Transition
         TOP : Bool := false;   // Zustand: Halbautomatisch/Ignoriere Transition
         ACK_S : Bool := false;   // Anforderung: Schritt quittieren, der an Parameter S_NO anliegt
         REG_S : Bool := false;   // Anforderung: Schritt registrieren, der an Parameter S_NO anliegt
         T_PREV : Bool := false;   // Anforderung: Vorherige gültige Transition am Parameter T_NO ausgeben
         T_NEXT : Bool := false;   // Anforderung: Nächste gültige Transition am Parameter T_NO ausgeben
         LOCK : Bool := true;   // Zustand: Interlockbearbeitung aktiviert
         SUP : Bool := true;   // Zustand: Supervisionsbearbeitung aktiviert
         ACKREQ : Bool := false;   // Zustand: Quittierung erforderlich
         SSKIP : Bool := false;   // Zustand: "Schritte überspringen" aktiviert
         OFF : Bool := false;   // Anforderung: Alle Schritte deaktivieren
         INIT : Bool := true;   // Anforderung: Kette in Initialzustand schalten
         HALT : Bool := false;   // Zustand: Kette schaltet nicht weiter
         TMS_HALT : Bool := false;   // Zustand: Alle internen Zeiten angehalten
         OPS_ZERO : Bool := false;   // Zustand: Alle mit N, L, D bearbeitete Operanden auf 0 gesetzt
         SACT_DISP : Bool := true;   // Zustand: Nur aktive Schritte anzeigen
         SEF_DISP : Bool := false;   // Zustand: Nur fehlerhafte und gestörte Schritte anzeigen
         SALL_DISP : Bool := false;   // Zustand: Alle Schritte anzeigen
         S_PREV : Bool := false;   // Anforderung: Vorherigen Schritt am Parameter S_NO ausgeben
         S_NEXT : Bool := false;   // Anforderung: Nächsten Schritt am Parameter S_NO ausgeben
         S_SELOK : Bool := false;   // Anforderung: Schrittnummer, die am Parameter S_SEL anliegt, am Parameter S_NO ausgeben
         S_ON : Bool := false;   // Anforderung: Schritt aktivieren, der am Parameter S_NO anliegt
         S_OFF : Bool := false;   // Anforderung: Schritt deaktivieren, der am Parameter S_NO anliegt
         T_PUSH : Bool := false;   // Anforderung: Schaltfreigabe für Transition
         REG : Bool := false;   // Anforderung: Alle Interlock- und Supervisionsfehler registrieren
         ACK : Bool := false;   // Anforderung: Alle Interlock- und Supervisionsfehler quittieren
         IL_PERM : Bool := false;   // Zustand: Permanente Bearbeitung aller Interlocks
         T_PERM : Bool := false;   // Zustand: Permanente Bearbeitung aller Transitionen
         ILP_MAN : Bool := false;   // Zustand: Permanente Bearbeitung aller Interlocks im Handbetrieb
      END_STRUCT;
      TICKS : Struct   // Zeittakte
         DELTA : Time := T#0ms;   // Zeitdifferenz zwischen zwei Zyklen
         OLD : Time := T#0ms;   // 10 ms Taktzählerstand im letzten Zyklus
         NEW : Time := T#0ms;   // 10 ms Taktzählerstand in diesem Zyklus
      END_STRUCT;
      SQ_FLAGS : Struct   // Kettenmerker
         ERR_FLT : Bool := false;   // Sammelfehler Interlock und Supervision
         ERROR : Bool := false;   // Sammelfehler Interlock
         FAULT : Bool := false;   // Sammelfehler Supervision
         RT_FAIL : Bool := false;   // Laufzeitfehler
         NO_SNO : Bool := false;   // Angeforderte Schrittnummer nicht gefunden
         NF_OFL : Bool := false;   // Überlauf: Zu viele Anforderungen ON oder OFF
         SA_OFL : Bool := false;   // Überlauf: Zu viele Schritte aktiv
         TV_OFL : Bool := false;   // Überlauf: Zu viele gültige Transitionen
         MSG_OFL : Bool := false;   // Überlauf: Nicht genügend Systemressourcen fü ALARM_S
         NO_SWI : Bool := false;   // Nicht Schalten in diesem Zyklus
         CYC_OP : Bool := false;   // Zyklische Bearbeitung der Kette nach Initialisierung
         AS_MSG : Bool := true;   // Meldungen zur Laufzeit durch Anweisung aktiviert oder deaktiviert
         AS_SEND : Bool := false;   // Meldungen von WR_USMSG senden oder nur in Diagnosepuffer eintragen
         SQ_BUSY : Bool := false;   // Interner Flankenmerker für Vorgangsbearbeitung
         SA_BUSY : Bool := false;   // Interner Flankenmerker für Vorgangsbearbeitung
         AS_SIG : Bool := false;   // Flankenmerker für Meldungen von Alarm_S und Alarm_SQ
      END_STRUCT;
      S_PTR : DWord := 16#450;
      S_PTR2 : DWord := 16#0;
      S_PTR3 : DWord := 16#D50;
      S_PTR4 : DWord := 16#D10;
      T_PTR : DWord := 16#CD0;
      C_AR2 : DWord := 16#0;
      M_FBDB : DWord := 16#8AE0000;
      M_SNO : Word := 16#4;
      M_EVID : Word := 16#0;
      M_EVIL : C_Alarm_s;
      M_EVSV : C_Alarm_s;
      M_EV : DWord := 16#C30;
      CRIT : Array[0..31] of Bool;
      S_START : Byte := 16#0;
      S_IDX : Byte := 16#0;
      S_INT : Int := 72;
      S_TMP : Byte := 16#0;
      T_START : Byte := 16#0;
      T_IDX : Byte := 16#0;
      T_TMP : Byte := 16#0;
      T_TMP2 : Byte := 16#00;
      TV_POT : Byte := 16#02;
      RETURN1 : Byte := 16#0;
      RETURN2 : Byte := 16#0;
      SINI : Array[0..2] of Byte;
      LSTT : Array[0..6] of Byte;
      ATAJ : Array[0..6] of Byte;
      ATAB : Array[0..6] of Byte;
      PSTT : Array[0..6] of Byte;
      NSTT : Array[0..6] of Byte;
      ASSJ : Array[0..6] of Byte;
      ASSB : Array[0..6] of Byte;
      PTTS : Array[0..6] of Byte;
      NTTS : Array[0..6] of Byte;
      PRE_CNT : Word := 16#2;
      POST_CNT : Word := 16#1;
      ADR_COND : Word := 16#0;
      MAX_TVAL : Byte := 16#1;
      MAX_SACT : Byte := 16#1;
      MAX_CRIT : Byte := 16#4;
      T_CNT : Byte := 16#6;
      SUP_CNT : Byte := 16#0;
      LOCK_CNT : Byte := 16#5;
      S_CNT : Byte := 16#6;
      SQ_CNT : Byte := 16#1;
      PRS_INPAR : DWord := 16#40000000;
      PRS_OUTPAR : DWord := 16#0;
      GC_FLAGS : Struct
         T_MACH : Byte := 16#EB;
         COND_ED : Byte := 16#E2;
         W_LEVEL : Byte := 16#D5;
         FB_IF : Byte := 16#FA;
         AS_MSG : Word := 16#404;
         SSB : Word := 16#108;
         DILG : Word := 16#27E;
         ADDR_T0 : Word := 16#1A;
         CRIT_AVAIL : Bool := false;
         SSKIP_AVAIL : Bool := true;
         SSKIP_ON : Bool := false;
         ACK_REQ : Bool := false;
         SYNC_AVAIL : Bool := true;
         ILP_MAN : Bool := false;
         SWM_LOCKED : Bool := false;
         SAVE_SW : Bool := true;
      END_STRUCT;
      G7_FBMARK : Byte := 16#3C;
      G7_RELEASE : Byte := 16#3C;
      G7_ID2 : Byte := 16#37;
      G7_ID1 : Byte := 16#47;
   END_VAR
   // SW_SQTS[0] := 16#1;
   // TVX[0] := 16#1;
   // TTX[0] := 16#1;
   // TSX[0] := 16#1;
   // S00X[0] := 16#1;
   // SOFFX[0] := 16#1;
   // SONX[0] := 16#1;
   // SAX[0] := 16#1;
   // SERRX[0] := 16#1;
   // SMX[0] := 16#1;
   // S0X[0] := 16#1;
   // S1X[0] := 16#1;
   // SINI[0] := 16#2;
   // SINI[1] := 16#1;
   // SINI[2] := 0;
   // LSTT[0] := 0;
   // LSTT[1] := 0;
   // LSTT[2] := 0;
   // LSTT[3] := 0;
   // LSTT[4] := 0;
   // LSTT[5] := 0;
   // LSTT[6] := 16#1;
   // ATAJ[0] := 0;
   // ATAJ[1] := 16#1;
   // ATAJ[2] := 16#2;
   // ATAJ[3] := 16#3;
   // ATAJ[4] := 16#4;
   // ATAJ[5] := 16#5;
   // ATAJ[6] := 16#6;
   // ATAB[0] := 0;
   // ATAB[1] := 16#1;
   // ATAB[2] := 16#2;
   // ATAB[3] := 16#3;
   // ATAB[4] := 16#4;
   // ATAB[5] := 16#5;
   // ATAB[6] := 16#6;
   // PSTT[0] := 0;
   // PSTT[1] := 16#1;
   // PSTT[2] := 16#2;
   // PSTT[3] := 16#3;
   // PSTT[4] := 16#4;
   // PSTT[5] := 16#5;
   // PSTT[6] := 16#6;
   // NSTT[0] := 16#1;
   // NSTT[1] := 16#2;
   // NSTT[2] := 16#3;
   // NSTT[3] := 16#4;
   // NSTT[4] := 16#5;
   // NSTT[5] := 16#6;
   // NSTT[6] := 16#1;
   // ASSJ[0] := 0;
   // ASSJ[1] := 16#1;
   // ASSJ[2] := 16#2;
   // ASSJ[3] := 16#3;
   // ASSJ[4] := 16#4;
   // ASSJ[5] := 16#5;
   // ASSJ[6] := 16#6;
   // ASSB[0] := 0;
   // ASSB[1] := 16#1;
   // ASSB[2] := 16#2;
   // ASSB[3] := 16#3;
   // ASSB[4] := 16#4;
   // ASSB[5] := 16#5;
   // ASSB[6] := 16#6;
   // PTTS[0] := 0;
   // PTTS[2] := 16#1;
   // PTTS[3] := 16#2;
   // PTTS[4] := 16#3;
   // PTTS[5] := 16#4;
   // PTTS[6] := 16#5;
   // NTTS[0] := 0;
   // NTTS[1] := 16#1;
   // NTTS[2] := 16#2;
   // NTTS[3] := 16#3;
   // NTTS[4] := 16#4;
   // NTTS[5] := 16#5;
   // NTTS[6] := 16#6;
BEGIN
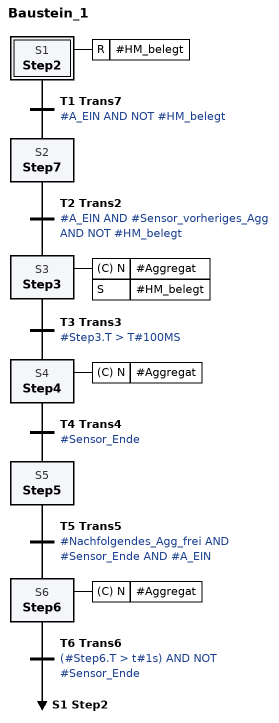
   // permanent pre-instructions
   NETWORK 1
      #HM_Agg_Frei := NOT #HM_belegt;
      #Aggregat_frei := NOT #HM_belegt;
   NETWORK 2
   TITLE = Ausgabe Schrittnummer
      #Schritt_Nummer := #S_DISPLAY;

   // sequencer 1
   INITIAL_STEP Step2:   // S1
      interlock C := NOT #A_NOT_HALT;
      // Warten auf Start
              R    #HM_belegt
   END_STEP
   TRANSITION Trans7 FROM Step2 TO Step7   // T1
      := #A_EIN AND NOT #HM_belegt;
   END_TRANSITION
   STEP Step4:   // S4
      interlock C := NOT #A_NOT_HALT;
      // Einfahrt bis Ende
      (C)     N    #Aggregat
   END_STEP
   TRANSITION Trans4 FROM Step4 TO Step5   // T4
      := #Sensor_Ende;
   END_TRANSITION
   STEP Step5:   // S5
      interlock C := NOT #A_NOT_HALT;
      // Warten auf Ausfahrt
   END_STEP
   TRANSITION Trans5 FROM Step5 TO Step6   // T5
      := #Nachfolgendes_Agg_frei AND #Sensor_Ende AND #A_EIN;
   END_TRANSITION
   STEP Step6:   // S6
      interlock C := NOT #A_NOT_HALT;
      // Ausfahrt bis Ende
      (C)     N    #Aggregat
   END_STEP
   TRANSITION Trans6 FROM Step6 TO Step2   // T6, jump
      := (#Step6.T > t#1s) AND NOT #Sensor_Ende;
   END_TRANSITION
   STEP Step3:   // S3
      interlock C := NOT #A_NOT_HALT;
      // Einfahrt Start
      (C)     N    #Aggregat
              S    #HM_belegt
   END_STEP
   TRANSITION Trans3 FROM Step3 TO Step4   // T3
      := #Step3.T > T#100MS;
   END_TRANSITION
   STEP Step7:   // S2
   END_STEP
   TRANSITION Trans2 FROM Step7 TO Step3   // T2
      := #A_EIN AND #Sensor_vorheriges_Agg AND NOT #HM_belegt;
   END_TRANSITION
END_FUNCTION_BLOCK